FUNCTION_BLOCK "Stanowisko_KB2"	// FB 4
//wyglad lini
//
//
//||||   ||     ||||   ||||
//|Z||  |O||    |W |   |S |
//||||   ||     ||||   ||||
//      
//      ||||
//      |B||
//      ||||
//
//Gdzie:
//-W-Winda
//-S-Shuttle
//-Z-ZPA(Segbert)
//-O-Obrotnica
//-B-Banda Backup
//
//
//Wersja 1.1
//-Dodanie mo¿liwosci poboru palety z Bandy backup (pisanie w trakcie)
//
//
//
AUTHOR : Kng
NAME : KB2
VERSION : 0.1
VAR
  KB2_Wylot_2 : FB 33;
  KB2_Obrotnica : FB 35;
  KB2_Uzbrajanie : FB 10;
  KB2_Winda : FB 37;
END_VAR
BEGIN
NETWORK
TITLE =
//Ten Network celowo jest wolny
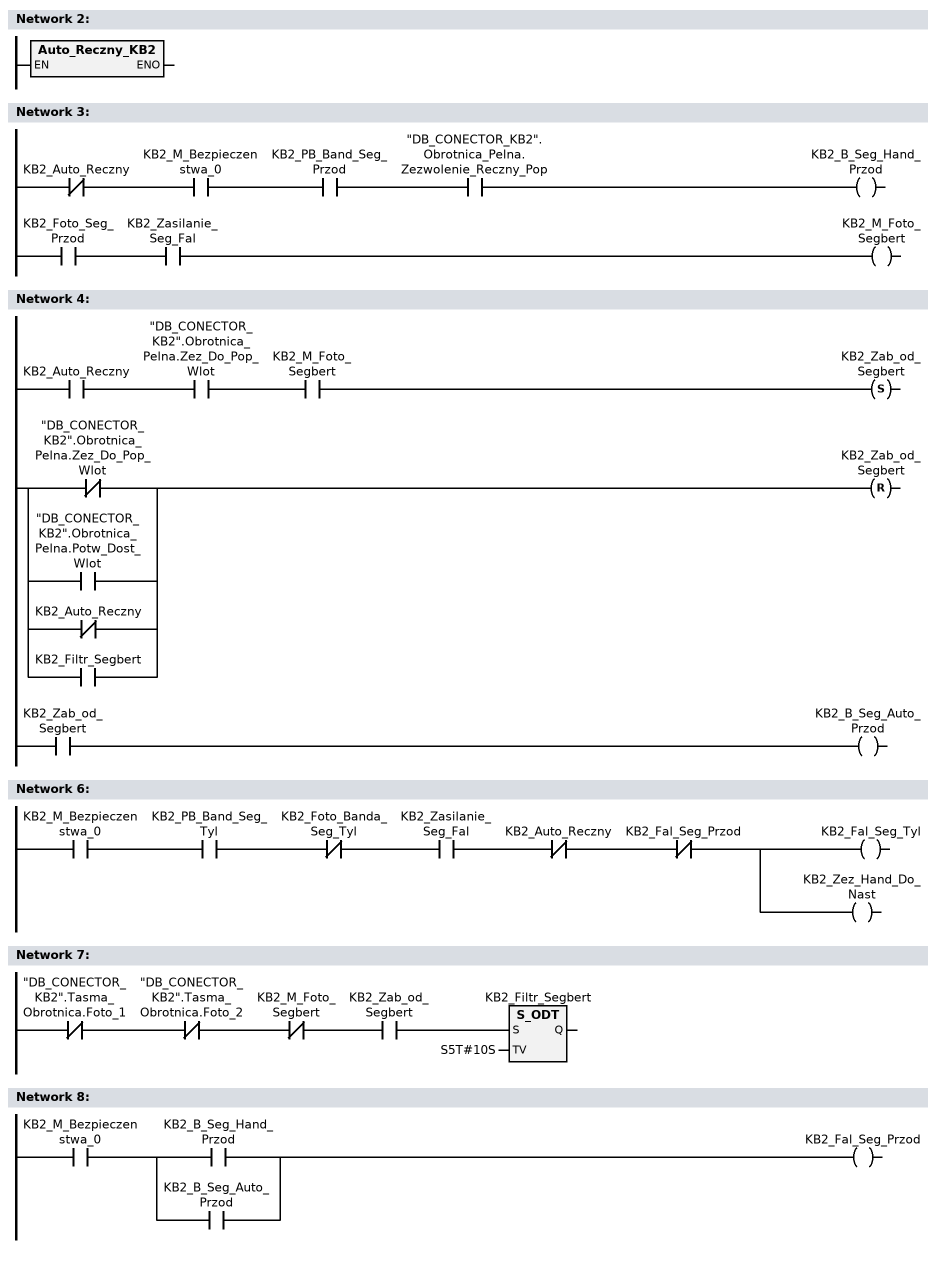
NETWORK
TITLE =
      CALL  "Auto_Reczny_KB2";
      NOP   0;
NETWORK
TITLE =
//Bity do Terminala
//
//Terminal_Palet                                   Szafa_Transport
//
//
//<-----------------------------------------------KB2_Fal_Seg_Przod (Q25.0)
//<-----------------------------------------------
//<-----------------------------------------------
//
//----------------------------------------------->KB2_Foto_Seg_Przod (I26.0)
//----------------------------------------------->
//----------------------------------------------->
//----------------------------------------------->
      AN    "KB2_Auto_Reczny";
      A     "KB2_M_Bezpieczenstwa_0";
      A     "KB2_PB_Band_Seg_Przod";
      A     "DB_CONECTOR_KB2".Obrotnica_Pelna.Zezwolenie_Reczny_Pop;
      =     "KB2_B_Seg_Hand_Przod";
//Wyjazd palety w automacie
      A     "KB2_Foto_Seg_Przod";
      A     "KB2_Zasilanie_Seg_Fal";
      =     "KB2_M_Foto_Segbert";
NETWORK
TITLE =
      A     "KB2_Auto_Reczny";
      A     "DB_CONECTOR_KB2".Obrotnica_Pelna.Zez_Do_Pop_Wlot;
      A     "KB2_M_Foto_Segbert";
      S     "KB2_Zab_od_Segbert";
      A(;
      ON    "DB_CONECTOR_KB2".Obrotnica_Pelna.Zez_Do_Pop_Wlot;
      O     "DB_CONECTOR_KB2".Obrotnica_Pelna.Potw_Dost_Wlot;
      ON    "KB2_Auto_Reczny";
      O     "KB2_Filtr_Segbert";
      );
      R     "KB2_Zab_od_Segbert";
      A     "KB2_Zab_od_Segbert";
      =     "KB2_B_Seg_Auto_Przod";
NETWORK
TITLE =
//Ten Network celowo jest wolny
NETWORK
TITLE =
//Segbert_Warunkowy tyl
      A     "KB2_M_Bezpieczenstwa_0";
      A     "KB2_PB_Band_Seg_Tyl";
      AN    "KB2_Foto_Banda_Seg_Tyl";
      A     "KB2_Zasilanie_Seg_Fal";
      AN    "KB2_Auto_Reczny";
      AN    "KB2_Fal_Seg_Przod";
      =     "KB2_Fal_Seg_Tyl";
      =     "KB2_Zez_Hand_Do_Nast";
NETWORK
TITLE =
      AN    "DB_CONECTOR_KB2".Tasma_Obrotnica.Foto_1;
      AN    "DB_CONECTOR_KB2".Tasma_Obrotnica.Foto_2;
      AN    "KB2_M_Foto_Segbert";
      A     "KB2_Zab_od_Segbert";
      L     S5T#10S;
      SD    "KB2_Filtr_Segbert";
      NOP   0;
      NOP   0;
      NOP   0;
      NOP   0;
NETWORK
TITLE =
//Jazda bandy Segbert do przodu
      A     "KB2_M_Bezpieczenstwa_0";
      A(;
      O     "KB2_B_Seg_Hand_Przod";
      O     "KB2_B_Seg_Auto_Przod";
      );
      =     "KB2_Fal_Seg_Przod";
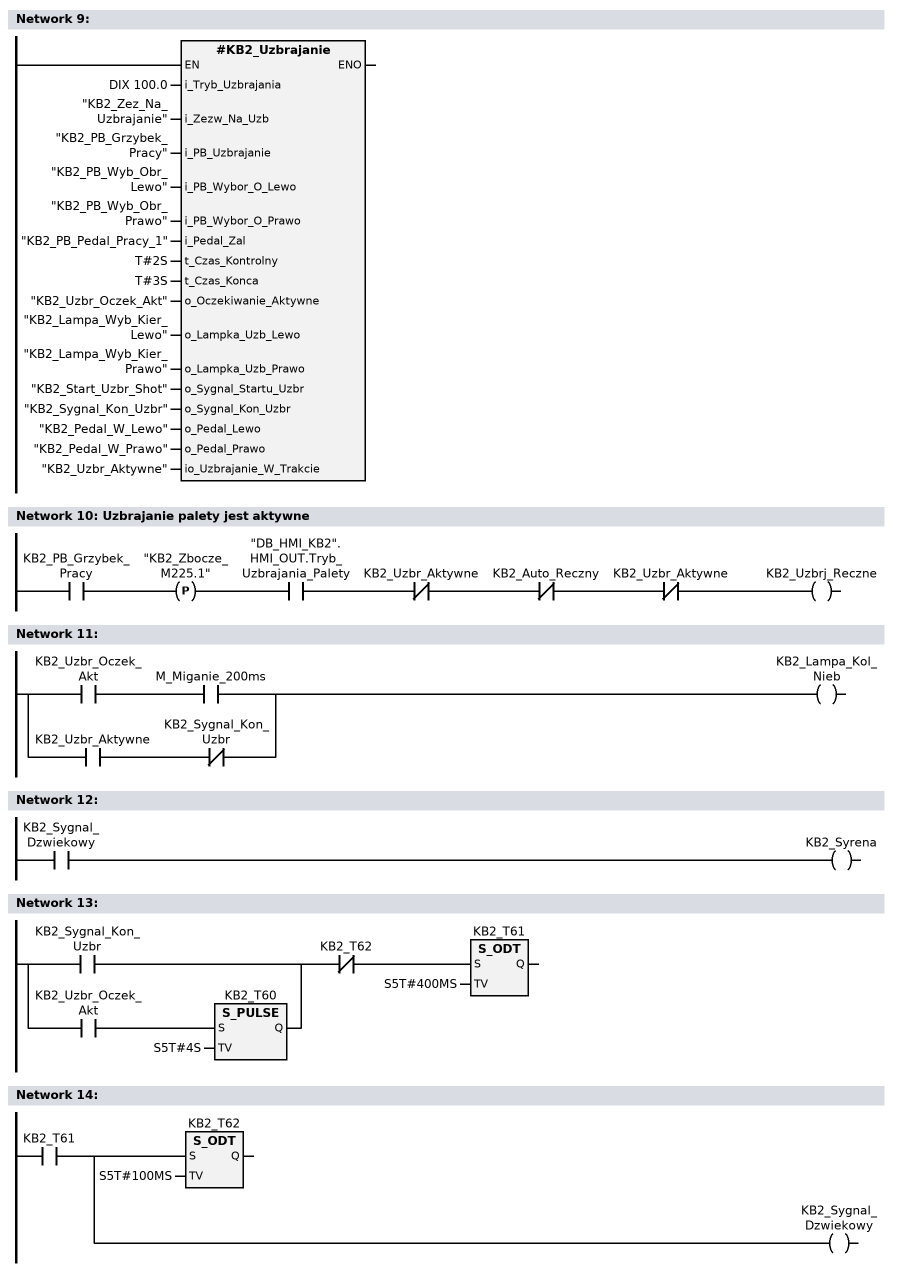
NETWORK
TITLE =
//Funkcja Uzbrajania
      CALL  #KB2_Uzbrajanie (
           i_Tryb_Uzbrajania        := DIX 100.0,
           i_Zezw_Na_Uzb            := "KB2_Zez_Na_Uzbrajanie",
           i_PB_Uzbrajanie          := "KB2_PB_Grzybek_Pracy",
           i_PB_Wybor_O_Lewo        := "KB2_PB_Wyb_Obr_Lewo",
           i_PB_Wybor_O_Prawo       := "KB2_PB_Wyb_Obr_Prawo",
           i_Pedal_Zal              := "KB2_PB_Pedal_Pracy_1",
           t_Czas_Kontrolny         := T#2S,
           t_Czas_Konca             := T#3S,
           o_Oczekiwanie_Aktywne    := "KB2_Uzbr_Oczek_Akt",
           o_Lampka_Uzb_Lewo        := "KB2_Lampa_Wyb_Kier_Lewo",
           o_Lampka_Uzb_Prawo       := "KB2_Lampa_Wyb_Kier_Prawo",
           o_Sygnal_Startu_Uzbr     := "KB2_Start_Uzbr_Shot",
           o_Sygnal_Kon_Uzbr        := "KB2_Sygnal_Kon_Uzbr",
           o_Pedal_Lewo             := "KB2_Pedal_W_Lewo",
           o_Pedal_Prawo            := "KB2_Pedal_W_Prawo",
           io_Uzbrajanie_W_Trakcie  := "KB2_Uzbr_Aktywne");
NETWORK
TITLE = Uzbrajanie palety jest aktywne
//Uzbrajanie reczne 
      A     "KB2_PB_Grzybek_Pracy";
      FP    "KB2_Zbocze_M225.1";
      A     "DB_HMI_KB2".HMI_OUT.Tryb_Uzbrajania_Palety;
      AN    "KB2_Uzbr_Aktywne";
      AN    "KB2_Auto_Reczny";
      AN    "KB2_Uzbr_Aktywne";
      =     "KB2_Uzbrj_Reczne";
NETWORK
TITLE =
//Lampka uzbrajania
//
      A     "KB2_Uzbr_Oczek_Akt";
      A     "M_Miganie_200ms";
      O;
      A     "KB2_Uzbr_Aktywne";
      AN    "KB2_Sygnal_Kon_Uzbr";
      =     "KB2_Lampa_Kol_Nieb";
NETWORK
TITLE =
//Sygnal dzwiekowy uzbrajania
//
      A     "KB2_Sygnal_Dzwiekowy";
      =     "KB2_Syrena";
NETWORK
TITLE =
//Tworzenie dzwieku
      A(;
      O     "KB2_Sygnal_Kon_Uzbr";
      O(;
      A     "KB2_Uzbr_Oczek_Akt";
      L     S5T#4S;
      SP    "KB2_T60";
      NOP   0;
      NOP   0;
      NOP   0;
      A     "KB2_T60";
      );
      );
      AN    "KB2_T62";
      L     S5T#400MS;
      SD    "KB2_T61";
      NOP   0;
      NOP   0;
      NOP   0;
      NOP   0;
NETWORK
TITLE =
      A     "KB2_T61";
      =     L 0.0;
      A     L 0.0;
      L     S5T#100MS;
      SD    "KB2_T62";
      NOP   0;
      NOP   0;
      NOP   0;
      NOP   0;
      A     L 0.0;
      BLD   102;
      =     "KB2_Sygnal_Dzwiekowy";
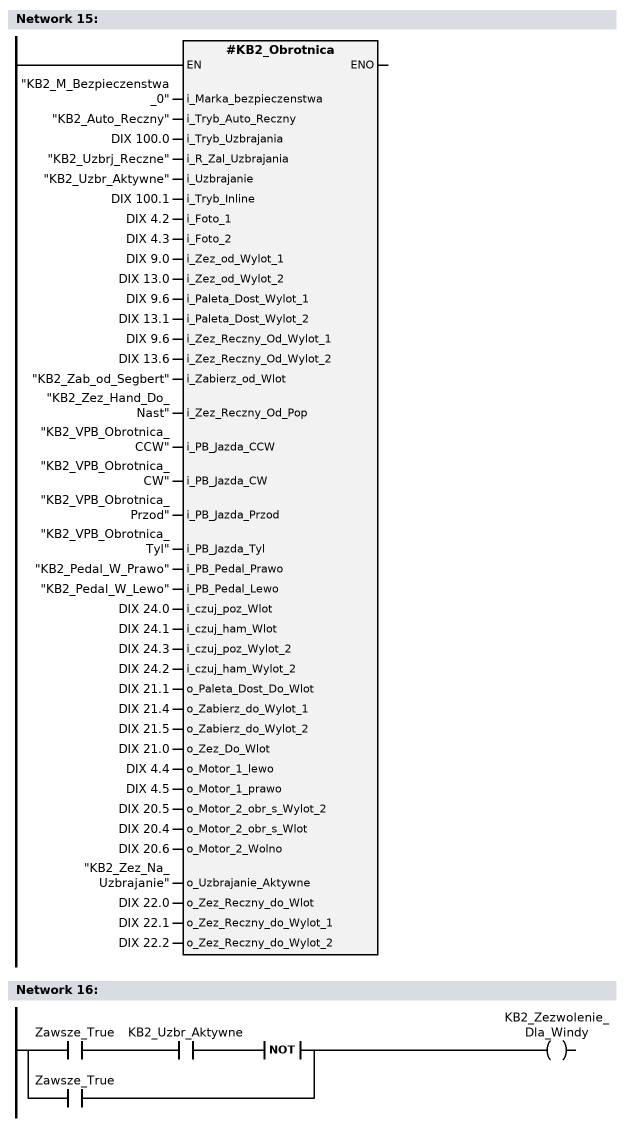
NETWORK
TITLE =
//Obrotnica z funkcja uzbrajania
      CALL  #KB2_Obrotnica (
           i_Marka_bezpieczenstwa   := "KB2_M_Bezpieczenstwa_0",
           i_Tryb_Auto_Reczny       := "KB2_Auto_Reczny",
           i_Tryb_Uzbrajania        := DIX 100.0,
           i_R_Zal_Uzbrajania       := "KB2_Uzbrj_Reczne",
           i_Uzbrajanie             := "KB2_Uzbr_Aktywne",
           i_Tryb_Inline            := DIX 100.1,
           i_Foto_1                 := DIX 4.2,
           i_Foto_2                 := DIX 4.3,
           i_Zez_od_Wylot_1         := DIX 9.0,
           i_Zez_od_Wylot_2         := DIX 13.0,
           i_Paleta_Dost_Wylot_1    := DIX 9.6,
           i_Paleta_Dost_Wylot_2    := DIX 13.1,
           i_Zez_Reczny_Od_Wylot_1  := DIX 9.6,
           i_Zez_Reczny_Od_Wylot_2  := DIX 13.6,
           i_Zabierz_od_Wlot        := "KB2_Zab_od_Segbert",
           i_Zez_Reczny_Od_Pop      := "KB2_Zez_Hand_Do_Nast",
           i_PB_Jazda_CCW           := "KB2_VPB_Obrotnica_CCW",
           i_PB_Jazda_CW            := "KB2_VPB_Obrotnica_CW",
           i_PB_Jazda_Przod         := "KB2_VPB_Obrotnica_Przod",
           i_PB_Jazda_Tyl           := "KB2_VPB_Obrotnica_Tyl",
           i_PB_Pedal_Prawo         := "KB2_Pedal_W_Prawo",
           i_PB_Pedal_Lewo          := "KB2_Pedal_W_Lewo",
           i_czuj_poz_Wlot          := DIX 24.0,
           i_czuj_ham_Wlot          := DIX 24.1,
           i_czuj_poz_Wylot_2       := DIX 24.3,
           i_czuj_ham_Wylot_2       := DIX 24.2,
           o_Paleta_Dost_Do_Wlot    := DIX 21.1,
           o_Zabierz_do_Wylot_1     := DIX 21.4,
           o_Zabierz_do_Wylot_2     := DIX 21.5,
           o_Zez_Do_Wlot            := DIX 21.0,
           o_Motor_1_lewo           := DIX 4.4,
           o_Motor_1_prawo          := DIX 4.5,
           o_Motor_2_obr_s_Wylot_2  := DIX 20.5,
           o_Motor_2_obr_s_Wlot     := DIX 20.4,
           o_Motor_2_Wolno          := DIX 20.6,
           o_Uzbrajanie_Aktywne     := "KB2_Zez_Na_Uzbrajanie",
           o_Zez_Reczny_do_Wlot     := DIX 22.0,
           o_Zez_Reczny_do_Wylot_1  := DIX 22.1,
           o_Zez_Reczny_do_Wylot_2  := DIX 22.2);
NETWORK
TITLE =
      A     "Zawsze_True";
      A     "KB2_Uzbr_Aktywne";
      NOT;
      O     "Zawsze_True";
      =     "KB2_Zezwolenie_Dla_Windy";
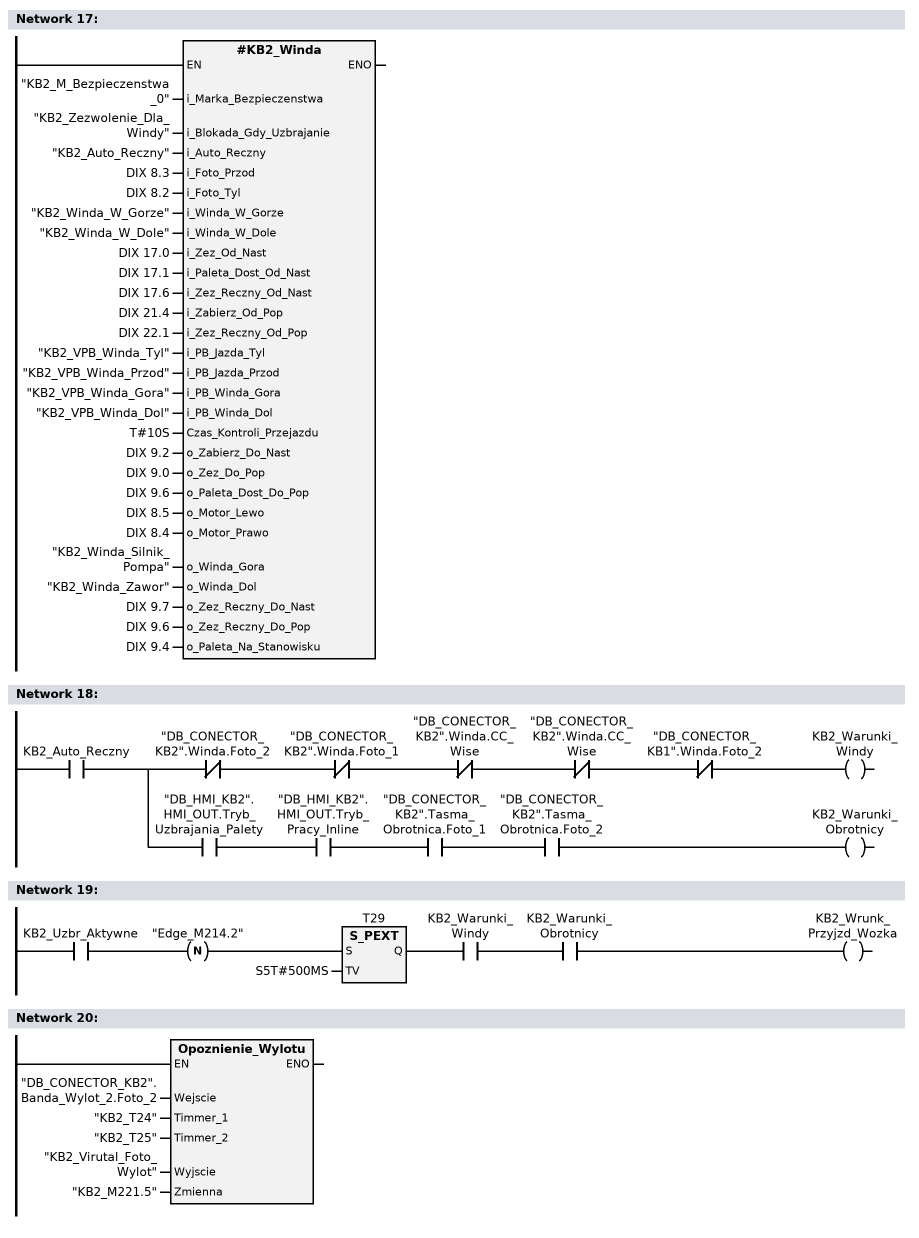
NETWORK
TITLE =
//Winda
      CALL  #KB2_Winda (
           i_Marka_Bezpieczenstwa   := "KB2_M_Bezpieczenstwa_0",
           i_Blokada_Gdy_Uzbrajanie := "KB2_Zezwolenie_Dla_Windy",
           i_Auto_Reczny            := "KB2_Auto_Reczny",
           i_Foto_Przod             := DIX 8.3,
           i_Foto_Tyl               := DIX 8.2,
           i_Winda_W_Gorze          := "KB2_Winda_W_Gorze",
           i_Winda_W_Dole           := "KB2_Winda_W_Dole",
           i_Zez_Od_Nast            := DIX 17.0,
           i_Paleta_Dost_Od_Nast    := DIX 17.1,
           i_Zez_Reczny_Od_Nast     := DIX 17.6,
           i_Zabierz_Od_Pop         := DIX 21.4,
           i_Zez_Reczny_Od_Pop      := DIX 22.1,
           i_PB_Jazda_Tyl           := "KB2_VPB_Winda_Tyl",
           i_PB_Jazda_Przod         := "KB2_VPB_Winda_Przod",
           i_PB_Winda_Gora          := "KB2_VPB_Winda_Gora",
           i_PB_Winda_Dol           := "KB2_VPB_Winda_Dol",
           Czas_Kontroli_Przejazdu  := T#10S,
           o_Zabierz_Do_Nast        := DIX 9.2,
           o_Zez_Do_Pop             := DIX 9.0,
           o_Paleta_Dost_Do_Pop     := DIX 9.6,
           o_Motor_Lewo             := DIX 8.5,
           o_Motor_Prawo            := DIX 8.4,
           o_Winda_Gora             := "KB2_Winda_Silnik_Pompa",
           o_Winda_Dol              := "KB2_Winda_Zawor",
           o_Zez_Reczny_Do_Nast     := DIX 9.7,
           o_Zez_Reczny_Do_Pop      := DIX 9.6,
           o_Paleta_Na_Stanowisku   := DIX 9.4);
NETWORK
TITLE =
//Warunkowa jazda wozka gdy konczone jest owijanie
//Warunki windy.
      A     "KB2_Auto_Reczny";
      =     L 0.0;
      A     L 0.0;
      AN    "DB_CONECTOR_KB2".Winda.Foto_2;
      AN    "DB_CONECTOR_KB2".Winda.Foto_1;
      AN    "DB_CONECTOR_KB2".Winda.CC_Wise;
      AN    "DB_CONECTOR_KB2".Winda.CC_Wise;
      AN    "DB_CONECTOR_KB1".Winda.Foto_2;
      =     "KB2_Warunki_Windy";
      A     L 0.0;
      A     "DB_HMI_KB2".HMI_OUT.Tryb_Uzbrajania_Palety;
      A     "DB_HMI_KB2".HMI_OUT.Tryb_Pracy_Inline;
      A     "DB_CONECTOR_KB2".Tasma_Obrotnica.Foto_1;
      A     "DB_CONECTOR_KB2".Tasma_Obrotnica.Foto_2;
      =     "KB2_Warunki_Obrotnicy";
NETWORK
TITLE =
//Warunki obrotnicy
      A(;
      A     "KB2_Uzbr_Aktywne";
      FN    "Edge_M214.2";
      L     S5T#500MS;
      SE    "T29";
      NOP   0;
      NOP   0;
      NOP   0;
      A     "T29";
      );
      A     "KB2_Warunki_Windy";
      A     "KB2_Warunki_Obrotnicy";
      =     "KB2_Wrunk_Przyjzd_Wozka";
NETWORK
TITLE =
//Opoznienie wylotu
      CALL  "Opoznienie_Wylotu" (
           Wejscie                  := "DB_CONECTOR_KB2".Banda_Wylot_2.Foto_2,
           Timmer_1                 := "KB2_T24",
           Timmer_2                 := "KB2_T25",
           Wyjscie                  := "KB2_Virutal_Foto_Wylot",
           Zmienna                  := "KB2_M221.5");
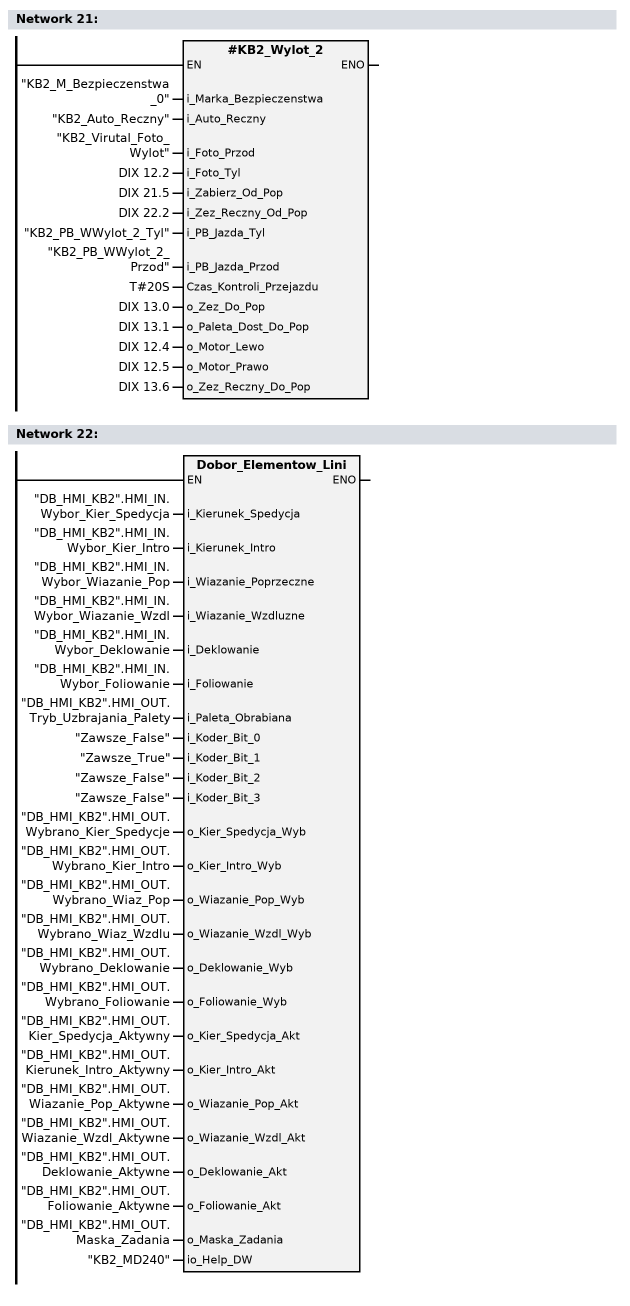
NETWORK
TITLE =
//Banda Wylot 2
      CALL  #KB2_Wylot_2 (
           i_Marka_Bezpieczenstwa   := "KB2_M_Bezpieczenstwa_0",
           i_Auto_Reczny            := "KB2_Auto_Reczny",
           i_Foto_Przod             := "KB2_Virutal_Foto_Wylot",
           i_Foto_Tyl               := DIX 12.2,
           i_Zabierz_Od_Pop         := DIX 21.5,
           i_Zez_Reczny_Od_Pop      := DIX 22.2,
           i_PB_Jazda_Tyl           := "KB2_PB_WWylot_2_Tyl",
           i_PB_Jazda_Przod         := "KB2_PB_WWylot_2_Przod",
           Czas_Kontroli_Przejazdu  := T#20S,
           o_Zez_Do_Pop             := DIX 13.0,
           o_Paleta_Dost_Do_Pop     := DIX 13.1,
           o_Motor_Lewo             := DIX 12.4,
           o_Motor_Prawo            := DIX 12.5,
           o_Zez_Reczny_Do_Pop      := DIX 13.6);
NETWORK
TITLE =
//fc400. Kod kolbus 2 to 2 .
      CALL  "Dobor_Elementow_Lini" (
           i_Kierunek_Spedycja      := "DB_HMI_KB2".HMI_IN.Wybor_Kier_Spedycja,
           i_Kierunek_Intro         := "DB_HMI_KB2".HMI_IN.Wybor_Kier_Intro,
           i_Wiazanie_Poprzeczne    := "DB_HMI_KB2".HMI_IN.Wybor_Wiazanie_Pop,
           i_Wiazanie_Wzdluzne      := "DB_HMI_KB2".HMI_IN.Wybor_Wiazanie_Wzdl,
           i_Deklowanie             := "DB_HMI_KB2".HMI_IN.Wybor_Deklowanie,
           i_Foliowanie             := "DB_HMI_KB2".HMI_IN.Wybor_Foliowanie,
           i_Paleta_Obrabiana       := "DB_HMI_KB2".HMI_OUT.Tryb_Uzbrajania_Palety,
           i_Koder_Bit_0            := "Zawsze_False",
           i_Koder_Bit_1            := "Zawsze_True",
           i_Koder_Bit_2            := "Zawsze_False",
           i_Koder_Bit_3            := "Zawsze_False",
           o_Kier_Spedycja_Wyb      := "DB_HMI_KB2".HMI_OUT.Wybrano_Kier_Spedycje,
           o_Kier_Intro_Wyb         := "DB_HMI_KB2".HMI_OUT.Wybrano_Kier_Intro,
           o_Wiazanie_Pop_Wyb       := "DB_HMI_KB2".HMI_OUT.Wybrano_Wiaz_Pop,
           o_Wiazanie_Wzdl_Wyb      := "DB_HMI_KB2".HMI_OUT.Wybrano_Wiaz_Wzdlu,
           o_Deklowanie_Wyb         := "DB_HMI_KB2".HMI_OUT.Wybrano_Deklowanie,
           o_Foliowanie_Wyb         := "DB_HMI_KB2".HMI_OUT.Wybrano_Foliowanie,
           o_Kier_Spedycja_Akt      := "DB_HMI_KB2".HMI_OUT.Kier_Spedycja_Aktywny,
           o_Kier_Intro_Akt         := "DB_HMI_KB2".HMI_OUT.Kierunek_Intro_Aktywny,
           o_Wiazanie_Pop_Akt       := "DB_HMI_KB2".HMI_OUT.Wiazanie_Pop_Aktywne,
           o_Wiazanie_Wzdl_Akt      := "DB_HMI_KB2".HMI_OUT.Wiazanie_Wzdl_Aktywne,
           o_Deklowanie_Akt         := "DB_HMI_KB2".HMI_OUT.Deklowanie_Aktywne,
           o_Foliowanie_Akt         := "DB_HMI_KB2".HMI_OUT.Foliowanie_Aktywne,
           o_Maska_Zadania          := "DB_HMI_KB2".HMI_OUT.Maska_Zadania,
           io_Help_DW               := "KB2_MD240");
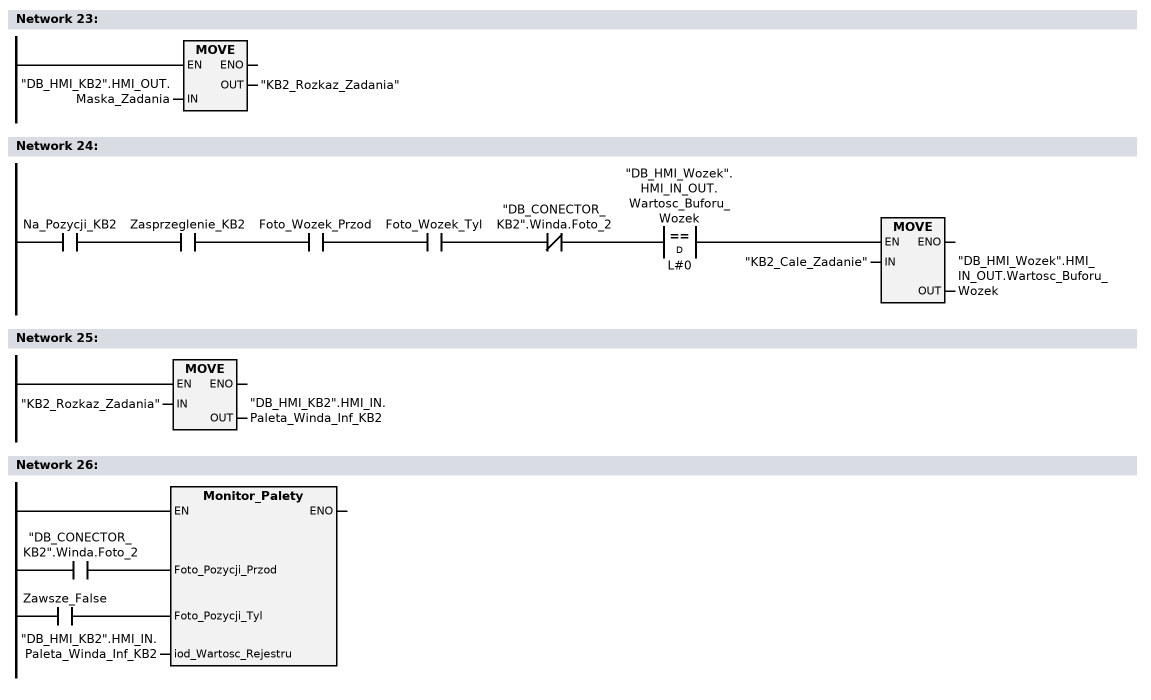
NETWORK
TITLE =
//Przeslanie maski do starszego slowa
      L     "DB_HMI_KB2".HMI_OUT.Maska_Zadania;
      T     "KB2_Rozkaz_Zadania";
      NOP   0;
NETWORK
TITLE =
//To jest wozek
//
      A     "Na_Pozycji_KB2";
      A     "Zasprzeglenie_KB2";
      A     "Foto_Wozek_Przod";
      A     "Foto_Wozek_Tyl";
      AN    "DB_CONECTOR_KB2".Winda.Foto_2;
      A(;
      L     "DB_HMI_Wozek".HMI_IN_OUT.Wartosc_Buforu_Wozek;
      L     L#0;
      ==D;
      );
      JNB   _001;
      L     "KB2_Cale_Zadanie";
      T     "DB_HMI_Wozek".HMI_IN_OUT.Wartosc_Buforu_Wozek;
_001: NOP   0;
NETWORK
TITLE =
      L     "KB2_Rozkaz_Zadania";
      T     "DB_HMI_KB2".HMI_IN.Paleta_Winda_Inf_KB2;
      NOP   0;
NETWORK
TITLE =
      A     "DB_CONECTOR_KB2".Winda.Foto_2;
      =     L 0.0;
      BLD   103;
      A     "Zawsze_False";
      =     L 0.1;
      BLD   103;
      CALL  "Monitor_Palety" (
           Foto_Pozycji_Przod       := L 0.0,
           Foto_Pozycji_Tyl         := L 0.1,
           iod_Wartosc_Rejestru     := "DB_HMI_KB2".HMI_IN.Paleta_Winda_Inf_KB2);
      NOP   0;
END_FUNCTION_BLOCK

FUNCTION_BLOCK "Stan_Intro_Odbieranie"	// FB 6
//Stanowisko intro Odbieranie
//Linia zlozona z 5 band odbierajacych
//
//
//BW B2 B3 B4 B4 B6
//===>
//
//5 band kierunek zwyczajny
VERSION : 0.1
VAR
  Banda_2 : FB 33;
  Banda_3 : FB 33;
  Banda_4 : FB 33;
  Banda_5 : FB 33;
  Banda_6 : FB 33;
END_VAR
VAR_TEMP
  help_bit_1 : BOOL ;
  Help_Reczny_Przod : BOOL ;
  Help_Reczny_Tyl : BOOL ;
END_VAR
BEGIN
NETWORK
TITLE =
//Ten Network celowo jest wolny
NETWORK
TITLE =
//Banda poprzednia jest wozek jezdny
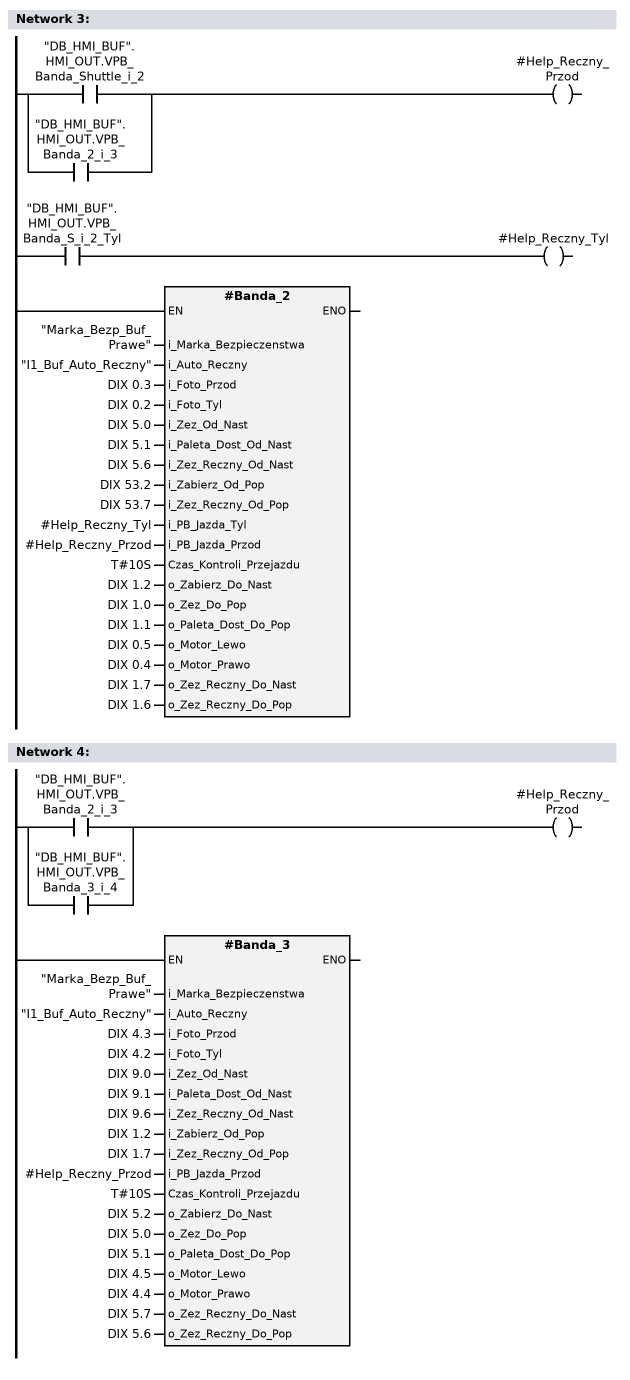
NETWORK
TITLE =
//Banda 2
      O     "DB_HMI_BUF".HMI_OUT.VPB_Banda_Shuttle_i_2;
      O     "DB_HMI_BUF".HMI_OUT.VPB_Banda_2_i_3;
      =     #Help_Reczny_Przod;
      O     "DB_HMI_BUF".HMI_OUT.VPB_Banda_S_i_2_Tyl;
      =     #Help_Reczny_Tyl;
      CALL  #Banda_2 (
           i_Marka_Bezpieczenstwa   := "Marka_Bezp_Buf_Prawe",
           i_Auto_Reczny            := "I1_Buf_Auto_Reczny",
           i_Foto_Przod             := DIX 0.3,
           i_Foto_Tyl               := DIX 0.2,
           i_Zez_Od_Nast            := DIX 5.0,
           i_Paleta_Dost_Od_Nast    := DIX 5.1,
           i_Zez_Reczny_Od_Nast     := DIX 5.6,
           i_Zabierz_Od_Pop         := DIX 53.2,
           i_Zez_Reczny_Od_Pop      := DIX 53.7,
           i_PB_Jazda_Tyl           := #Help_Reczny_Tyl,
           i_PB_Jazda_Przod         := #Help_Reczny_Przod,
           Czas_Kontroli_Przejazdu  := T#10S,
           o_Zabierz_Do_Nast        := DIX 1.2,
           o_Zez_Do_Pop             := DIX 1.0,
           o_Paleta_Dost_Do_Pop     := DIX 1.1,
           o_Motor_Lewo             := DIX 0.5,
           o_Motor_Prawo            := DIX 0.4,
           o_Zez_Reczny_Do_Nast     := DIX 1.7,
           o_Zez_Reczny_Do_Pop      := DIX 1.6);
NETWORK
TITLE =
//Banda 3
      O     "DB_HMI_BUF".HMI_OUT.VPB_Banda_2_i_3;
      O     "DB_HMI_BUF".HMI_OUT.VPB_Banda_3_i_4;
      =     #Help_Reczny_Przod;
      CALL  #Banda_3 (
           i_Marka_Bezpieczenstwa   := "Marka_Bezp_Buf_Prawe",
           i_Auto_Reczny            := "I1_Buf_Auto_Reczny",
           i_Foto_Przod             := DIX 4.3,
           i_Foto_Tyl               := DIX 4.2,
           i_Zez_Od_Nast            := DIX 9.0,
           i_Paleta_Dost_Od_Nast    := DIX 9.1,
           i_Zez_Reczny_Od_Nast     := DIX 9.6,
           i_Zabierz_Od_Pop         := DIX 1.2,
           i_Zez_Reczny_Od_Pop      := DIX 1.7,
           i_PB_Jazda_Przod         := #Help_Reczny_Przod,
           Czas_Kontroli_Przejazdu  := T#10S,
           o_Zabierz_Do_Nast        := DIX 5.2,
           o_Zez_Do_Pop             := DIX 5.0,
           o_Paleta_Dost_Do_Pop     := DIX 5.1,
           o_Motor_Lewo             := DIX 4.5,
           o_Motor_Prawo            := DIX 4.4,
           o_Zez_Reczny_Do_Nast     := DIX 5.7,
           o_Zez_Reczny_Do_Pop      := DIX 5.6);
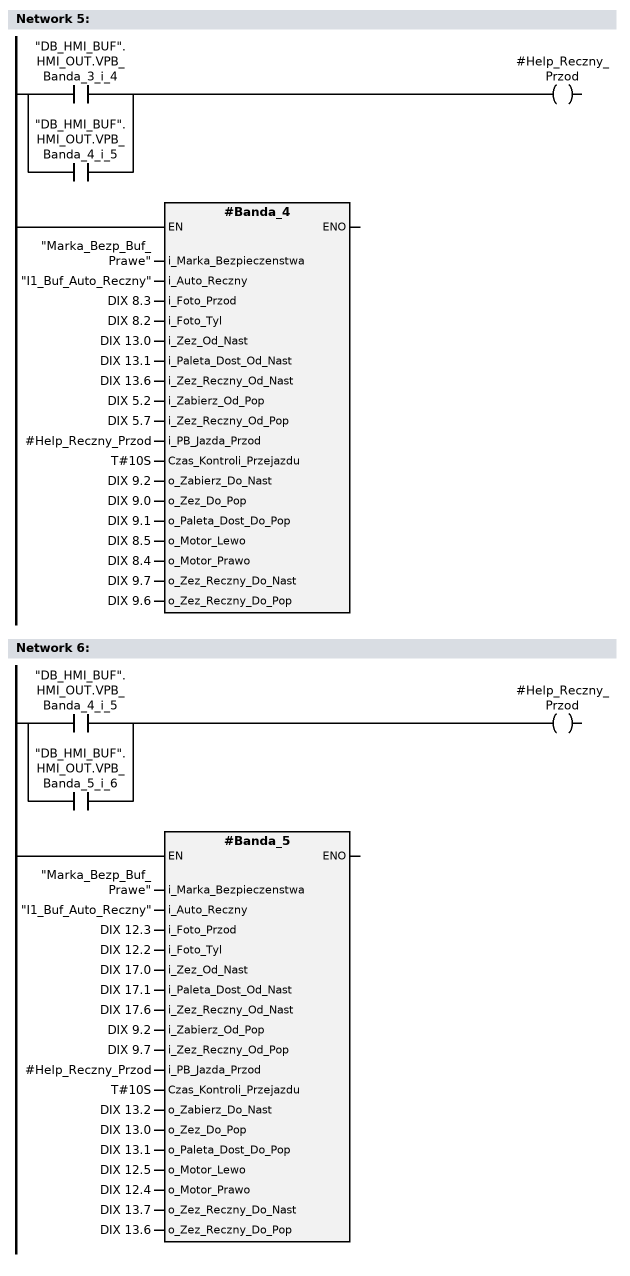
NETWORK
TITLE =
//Banda 4
      O     "DB_HMI_BUF".HMI_OUT.VPB_Banda_3_i_4;
      O     "DB_HMI_BUF".HMI_OUT.VPB_Banda_4_i_5;
      =     #Help_Reczny_Przod;
      CALL  #Banda_4 (
           i_Marka_Bezpieczenstwa   := "Marka_Bezp_Buf_Prawe",
           i_Auto_Reczny            := "I1_Buf_Auto_Reczny",
           i_Foto_Przod             := DIX 8.3,
           i_Foto_Tyl               := DIX 8.2,
           i_Zez_Od_Nast            := DIX 13.0,
           i_Paleta_Dost_Od_Nast    := DIX 13.1,
           i_Zez_Reczny_Od_Nast     := DIX 13.6,
           i_Zabierz_Od_Pop         := DIX 5.2,
           i_Zez_Reczny_Od_Pop      := DIX 5.7,
           i_PB_Jazda_Przod         := #Help_Reczny_Przod,
           Czas_Kontroli_Przejazdu  := T#10S,
           o_Zabierz_Do_Nast        := DIX 9.2,
           o_Zez_Do_Pop             := DIX 9.0,
           o_Paleta_Dost_Do_Pop     := DIX 9.1,
           o_Motor_Lewo             := DIX 8.5,
           o_Motor_Prawo            := DIX 8.4,
           o_Zez_Reczny_Do_Nast     := DIX 9.7,
           o_Zez_Reczny_Do_Pop      := DIX 9.6);
NETWORK
TITLE =
//Banda 5
      O     "DB_HMI_BUF".HMI_OUT.VPB_Banda_4_i_5;
      O     "DB_HMI_BUF".HMI_OUT.VPB_Banda_5_i_6;
      =     #Help_Reczny_Przod;
      CALL  #Banda_5 (
           i_Marka_Bezpieczenstwa   := "Marka_Bezp_Buf_Prawe",
           i_Auto_Reczny            := "I1_Buf_Auto_Reczny",
           i_Foto_Przod             := DIX 12.3,
           i_Foto_Tyl               := DIX 12.2,
           i_Zez_Od_Nast            := DIX 17.0,
           i_Paleta_Dost_Od_Nast    := DIX 17.1,
           i_Zez_Reczny_Od_Nast     := DIX 17.6,
           i_Zabierz_Od_Pop         := DIX 9.2,
           i_Zez_Reczny_Od_Pop      := DIX 9.7,
           i_PB_Jazda_Przod         := #Help_Reczny_Przod,
           Czas_Kontroli_Przejazdu  := T#10S,
           o_Zabierz_Do_Nast        := DIX 13.2,
           o_Zez_Do_Pop             := DIX 13.0,
           o_Paleta_Dost_Do_Pop     := DIX 13.1,
           o_Motor_Lewo             := DIX 12.5,
           o_Motor_Prawo            := DIX 12.4,
           o_Zez_Reczny_Do_Nast     := DIX 13.7,
           o_Zez_Reczny_Do_Pop      := DIX 13.6);
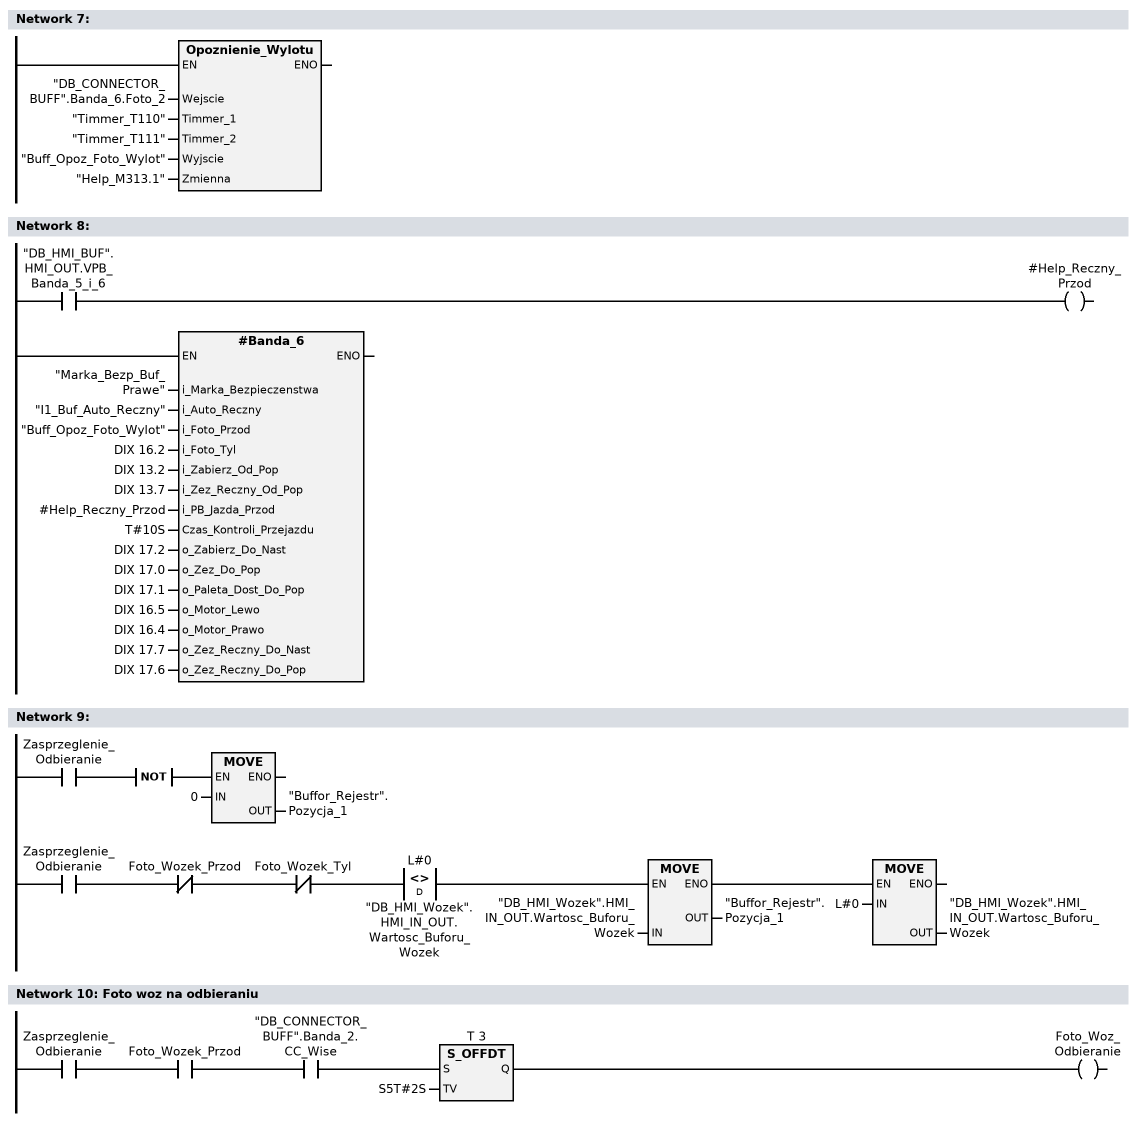
NETWORK
TITLE =
      CALL  "Opoznienie_Wylotu" (
           Wejscie                  := "DB_CONNECTOR_BUFF".Banda_6.Foto_2,
           Timmer_1                 := "Timmer_T110",
           Timmer_2                 := "Timmer_T111",
           Wyjscie                  := "Buff_Opoz_Foto_Wylot",
           Zmienna                  := "Help_M313.1");
NETWORK
TITLE =
//Banda 6
      O     "DB_HMI_BUF".HMI_OUT.VPB_Banda_5_i_6;
      =     #Help_Reczny_Przod;
      CALL  #Banda_6 (
           i_Marka_Bezpieczenstwa   := "Marka_Bezp_Buf_Prawe",
           i_Auto_Reczny            := "I1_Buf_Auto_Reczny",
           i_Foto_Przod             := "Buff_Opoz_Foto_Wylot",
           i_Foto_Tyl               := DIX 16.2,
           i_Zabierz_Od_Pop         := DIX 13.2,
           i_Zez_Reczny_Od_Pop      := DIX 13.7,
           i_PB_Jazda_Przod         := #Help_Reczny_Przod,
           Czas_Kontroli_Przejazdu  := T#10S,
           o_Zabierz_Do_Nast        := DIX 17.2,
           o_Zez_Do_Pop             := DIX 17.0,
           o_Paleta_Dost_Do_Pop     := DIX 17.1,
           o_Motor_Lewo             := DIX 16.5,
           o_Motor_Prawo            := DIX 16.4,
           o_Zez_Reczny_Do_Nast     := DIX 17.7,
           o_Zez_Reczny_Do_Pop      := DIX 17.6);
NETWORK
TITLE =
      A     "Zasprzeglenie_Odbieranie";
      =     L 1.0;
      A(;
      A     L 1.0;
      AN    "Foto_Wozek_Przod";
      AN    "Foto_Wozek_Tyl";
      A(;
      L     L#0;
      L     "DB_HMI_Wozek".HMI_IN_OUT.Wartosc_Buforu_Wozek;
      <>D;
      );
      JNB   _001;
      L     "DB_HMI_Wozek".HMI_IN_OUT.Wartosc_Buforu_Wozek;
      T     "Buffor_Rejestr".Pozycja_1;
      SET;
      SAVE;
      CLR;
_001: A     BR;
      );
      JNB   _002;
      L     L#0;
      T     "DB_HMI_Wozek".HMI_IN_OUT.Wartosc_Buforu_Wozek;
_002: NOP   0;
      A     L 1.0;
      NOT;
      JNB   _003;
      L     0;
      T     "Buffor_Rejestr".Pozycja_1;
_003: NOP   0;
NETWORK
TITLE = Foto woz na odbieraniu
      A     "Zasprzeglenie_Odbieranie";
      A     "Foto_Wozek_Przod";
      A     "DB_CONNECTOR_BUFF".Banda_2.CC_Wise;
      L     S5T#2S;
      SF    T 3;
      NOP   0;
      NOP   0;
      NOP   0;
      A     T 3;
      =     "Foto_Woz_Odbieranie";
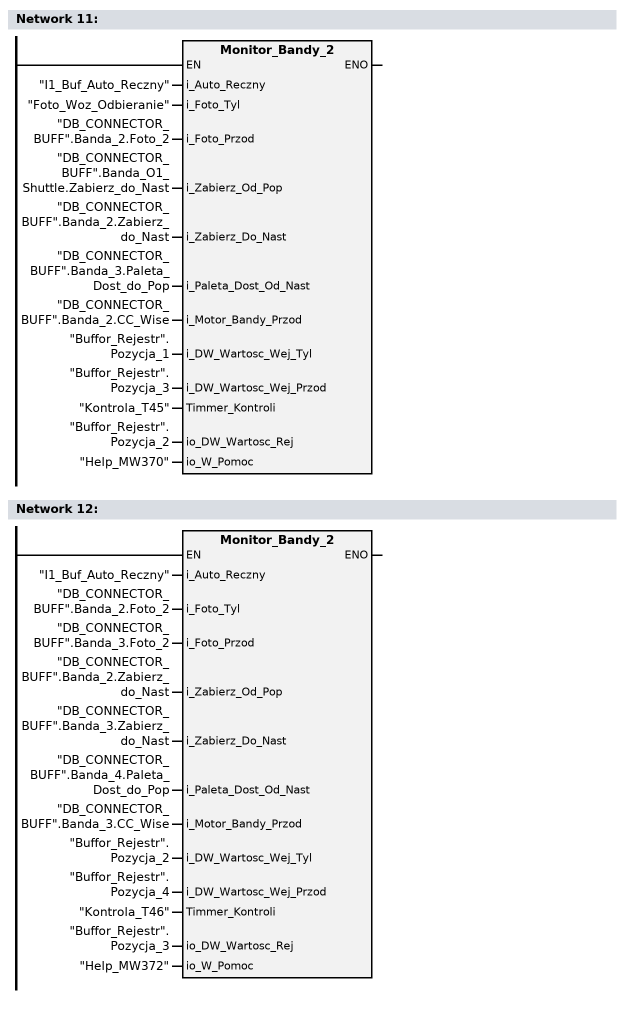
NETWORK
TITLE =
//Monitoring band 2
      CALL  "Monitor_Bandy_2" (
           i_Auto_Reczny            := "I1_Buf_Auto_Reczny",
           i_Foto_Tyl               := "Foto_Woz_Odbieranie",
           i_Foto_Przod             := "DB_CONNECTOR_BUFF".Banda_2.Foto_2,
           i_Zabierz_Od_Pop         := "DB_CONNECTOR_BUFF".Banda_O1_Shuttle.Zabierz_do_Nast,
           i_Zabierz_Do_Nast        := "DB_CONNECTOR_BUFF".Banda_2.Zabierz_do_Nast,
           i_Paleta_Dost_Od_Nast    := "DB_CONNECTOR_BUFF".Banda_3.Paleta_Dost_do_Pop,
           i_Motor_Bandy_Przod      := "DB_CONNECTOR_BUFF".Banda_2.CC_Wise,
           i_DW_Wartosc_Wej_Tyl     := "Buffor_Rejestr".Pozycja_1,
           i_DW_Wartosc_Wej_Przod   := "Buffor_Rejestr".Pozycja_3,
           Timmer_Kontroli          := "Kontrola_T45",
           io_DW_Wartosc_Rej        := "Buffor_Rejestr".Pozycja_2,
           io_W_Pomoc               := "Help_MW370");
NETWORK
TITLE =
//Monitoring band 3
      CALL  "Monitor_Bandy_2" (
           i_Auto_Reczny            := "I1_Buf_Auto_Reczny",
           i_Foto_Tyl               := "DB_CONNECTOR_BUFF".Banda_2.Foto_2,
           i_Foto_Przod             := "DB_CONNECTOR_BUFF".Banda_3.Foto_2,
           i_Zabierz_Od_Pop         := "DB_CONNECTOR_BUFF".Banda_2.Zabierz_do_Nast,
           i_Zabierz_Do_Nast        := "DB_CONNECTOR_BUFF".Banda_3.Zabierz_do_Nast,
           i_Paleta_Dost_Od_Nast    := "DB_CONNECTOR_BUFF".Banda_4.Paleta_Dost_do_Pop,
           i_Motor_Bandy_Przod      := "DB_CONNECTOR_BUFF".Banda_3.CC_Wise,
           i_DW_Wartosc_Wej_Tyl     := "Buffor_Rejestr".Pozycja_2,
           i_DW_Wartosc_Wej_Przod   := "Buffor_Rejestr".Pozycja_4,
           Timmer_Kontroli          := "Kontrola_T46",
           io_DW_Wartosc_Rej        := "Buffor_Rejestr".Pozycja_3,
           io_W_Pomoc               := "Help_MW372");
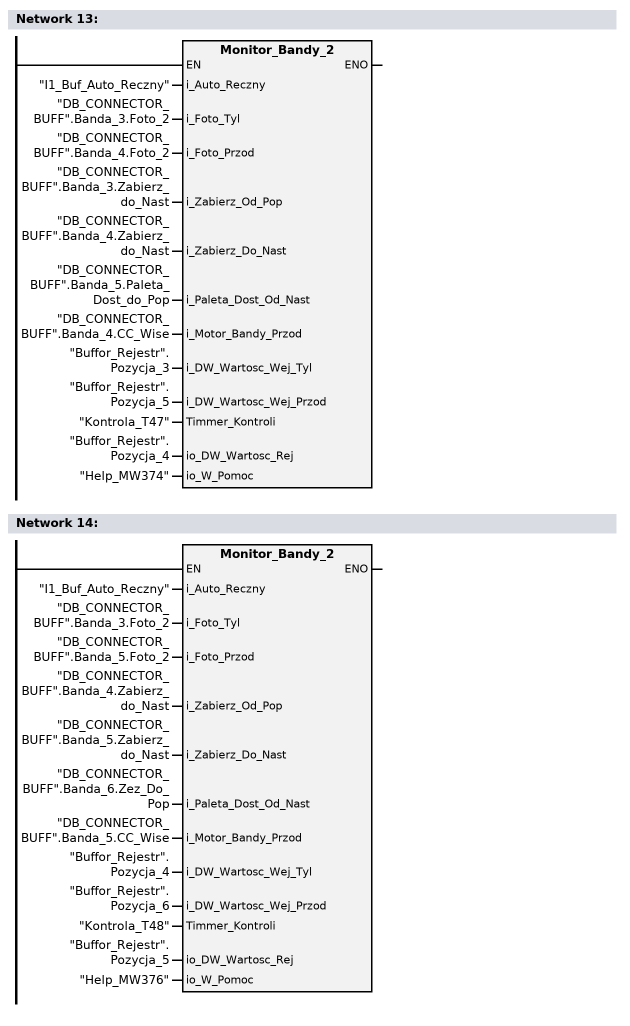
NETWORK
TITLE =
//Monitoring band 4
      CALL  "Monitor_Bandy_2" (
           i_Auto_Reczny            := "I1_Buf_Auto_Reczny",
           i_Foto_Tyl               := "DB_CONNECTOR_BUFF".Banda_3.Foto_2,
           i_Foto_Przod             := "DB_CONNECTOR_BUFF".Banda_4.Foto_2,
           i_Zabierz_Od_Pop         := "DB_CONNECTOR_BUFF".Banda_3.Zabierz_do_Nast,
           i_Zabierz_Do_Nast        := "DB_CONNECTOR_BUFF".Banda_4.Zabierz_do_Nast,
           i_Paleta_Dost_Od_Nast    := "DB_CONNECTOR_BUFF".Banda_5.Paleta_Dost_do_Pop,
           i_Motor_Bandy_Przod      := "DB_CONNECTOR_BUFF".Banda_4.CC_Wise,
           i_DW_Wartosc_Wej_Tyl     := "Buffor_Rejestr".Pozycja_3,
           i_DW_Wartosc_Wej_Przod   := "Buffor_Rejestr".Pozycja_5,
           Timmer_Kontroli          := "Kontrola_T47",
           io_DW_Wartosc_Rej        := "Buffor_Rejestr".Pozycja_4,
           io_W_Pomoc               := "Help_MW374");
NETWORK
TITLE =
//Monitoring band 5
//
      CALL  "Monitor_Bandy_2" (
           i_Auto_Reczny            := "I1_Buf_Auto_Reczny",
           i_Foto_Tyl               := "DB_CONNECTOR_BUFF".Banda_3.Foto_2,
           i_Foto_Przod             := "DB_CONNECTOR_BUFF".Banda_5.Foto_2,
           i_Zabierz_Od_Pop         := "DB_CONNECTOR_BUFF".Banda_4.Zabierz_do_Nast,
           i_Zabierz_Do_Nast        := "DB_CONNECTOR_BUFF".Banda_5.Zabierz_do_Nast,
           i_Paleta_Dost_Od_Nast    := "DB_CONNECTOR_BUFF".Banda_6.Zez_Do_Pop,
           i_Motor_Bandy_Przod      := "DB_CONNECTOR_BUFF".Banda_5.CC_Wise,
           i_DW_Wartosc_Wej_Tyl     := "Buffor_Rejestr".Pozycja_4,
           i_DW_Wartosc_Wej_Przod   := "Buffor_Rejestr".Pozycja_6,
           Timmer_Kontroli          := "Kontrola_T48",
           io_DW_Wartosc_Rej        := "Buffor_Rejestr".Pozycja_5,
           io_W_Pomoc               := "Help_MW376");
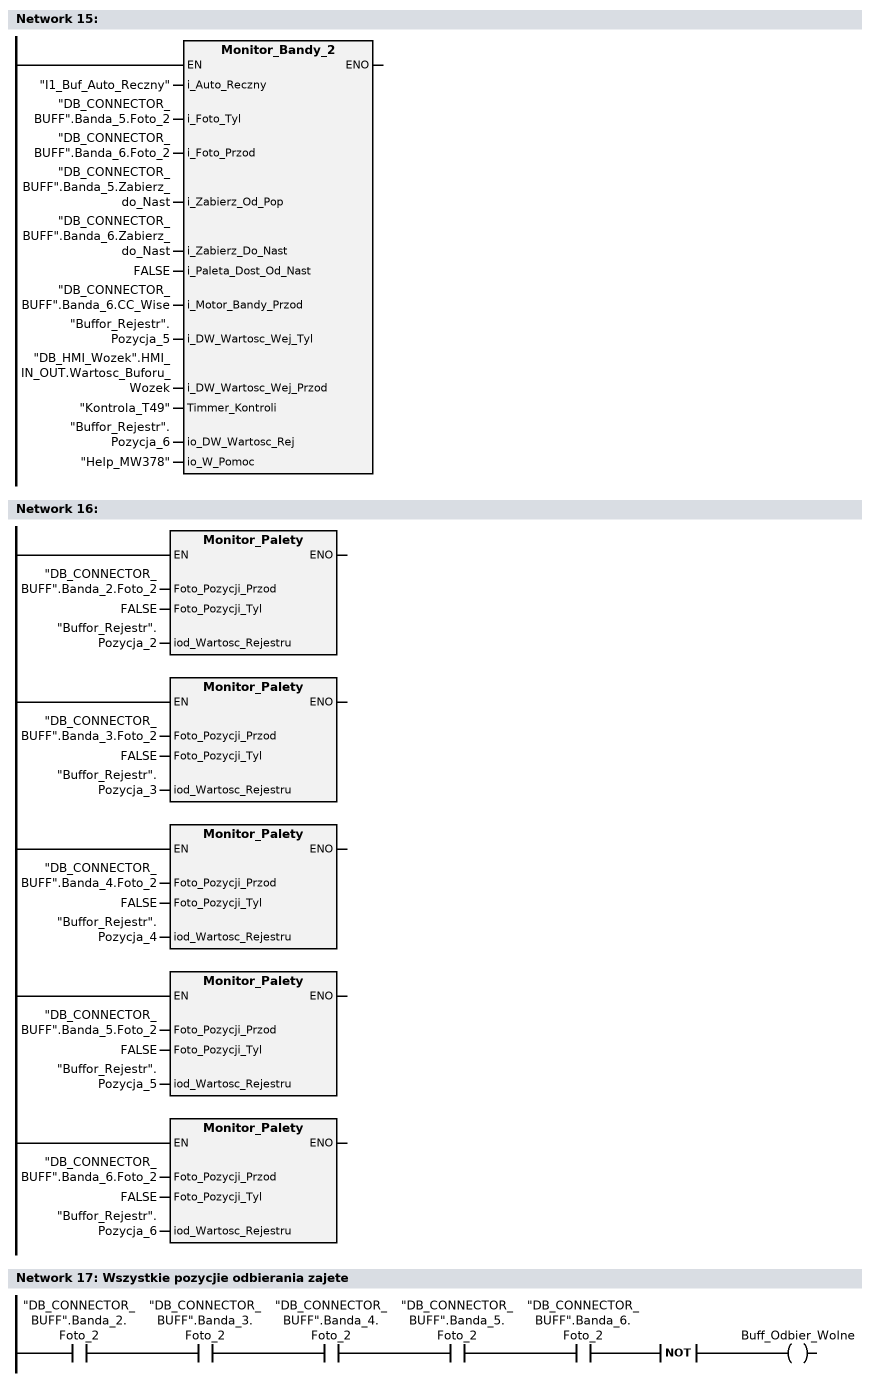
NETWORK
TITLE =
//Monitoring band 6
      CALL  "Monitor_Bandy_2" (
           i_Auto_Reczny            := "I1_Buf_Auto_Reczny",
           i_Foto_Tyl               := "DB_CONNECTOR_BUFF".Banda_5.Foto_2,
           i_Foto_Przod             := "DB_CONNECTOR_BUFF".Banda_6.Foto_2,
           i_Zabierz_Od_Pop         := "DB_CONNECTOR_BUFF".Banda_5.Zabierz_do_Nast,
           i_Zabierz_Do_Nast        := "DB_CONNECTOR_BUFF".Banda_6.Zabierz_do_Nast,
           i_Paleta_Dost_Od_Nast    := FALSE,
           i_Motor_Bandy_Przod      := "DB_CONNECTOR_BUFF".Banda_6.CC_Wise,
           i_DW_Wartosc_Wej_Tyl     := "Buffor_Rejestr".Pozycja_5,
           i_DW_Wartosc_Wej_Przod   := "DB_HMI_Wozek".HMI_IN_OUT.Wartosc_Buforu_Wozek,
           Timmer_Kontroli          := "Kontrola_T49",
           io_DW_Wartosc_Rej        := "Buffor_Rejestr".Pozycja_6,
           io_W_Pomoc               := "Help_MW378");
NETWORK
TITLE =
//Zaznaczenie czy jest paleta
      CALL  "Monitor_Palety" (
           Foto_Pozycji_Przod       := "DB_CONNECTOR_BUFF".Banda_2.Foto_2,
           Foto_Pozycji_Tyl         := FALSE,
           iod_Wartosc_Rejestru     := "Buffor_Rejestr".Pozycja_2);
      CALL  "Monitor_Palety" (
           Foto_Pozycji_Przod       := "DB_CONNECTOR_BUFF".Banda_3.Foto_2,
           Foto_Pozycji_Tyl         := FALSE,
           iod_Wartosc_Rejestru     := "Buffor_Rejestr".Pozycja_3);
      CALL  "Monitor_Palety" (
           Foto_Pozycji_Przod       := "DB_CONNECTOR_BUFF".Banda_4.Foto_2,
           Foto_Pozycji_Tyl         := FALSE,
           iod_Wartosc_Rejestru     := "Buffor_Rejestr".Pozycja_4);
      CALL  "Monitor_Palety" (
           Foto_Pozycji_Przod       := "DB_CONNECTOR_BUFF".Banda_5.Foto_2,
           Foto_Pozycji_Tyl         := FALSE,
           iod_Wartosc_Rejestru     := "Buffor_Rejestr".Pozycja_5);
      CALL  "Monitor_Palety" (
           Foto_Pozycji_Przod       := "DB_CONNECTOR_BUFF".Banda_6.Foto_2,
           Foto_Pozycji_Tyl         := FALSE,
           iod_Wartosc_Rejestru     := "Buffor_Rejestr".Pozycja_6);
NETWORK
TITLE = Wszystkie pozycjie odbierania zajete
//Sprawdzenie czy wszystkie pozycje sa zajete
      A     "DB_CONNECTOR_BUFF".Banda_2.Foto_2;
      A     "DB_CONNECTOR_BUFF".Banda_3.Foto_2;
      A     "DB_CONNECTOR_BUFF".Banda_4.Foto_2;
      A     "DB_CONNECTOR_BUFF".Banda_5.Foto_2;
      A     "DB_CONNECTOR_BUFF".Banda_6.Foto_2;
      NOT;
      =     "Buff_Odbier_Wolne";
END_FUNCTION_BLOCK

FUNCTION_BLOCK "Stan_Intro_Pob_I1"	// FB 7
//Stanowisko intro Pobieranie
//Linia zlozona z 5 band odbierajacych
//
//
//BW B16 B15 B14 B13 B12 
//             <===
//
//5 band kierunek zanegowany
VERSION : 0.1
VAR
  Banda_12 : FB 33;
  Banda_13 : FB 33;
  Banda_14 : FB 33;
  Banda_15 : FB 33;
  Banda_16 : FB 33;
END_VAR
VAR_TEMP
  Help_Bit_1 : BOOL ;
  Help_Reczny_Przod : BOOL ;
  Help_Reczny_Tyl : BOOL ;
  Help_int : INT ;
  Help_Dword : DWORD ;
  Help_INT_1 : DINT ;
END_VAR
BEGIN
NETWORK
TITLE =
//Ten Network celowo jest wolny
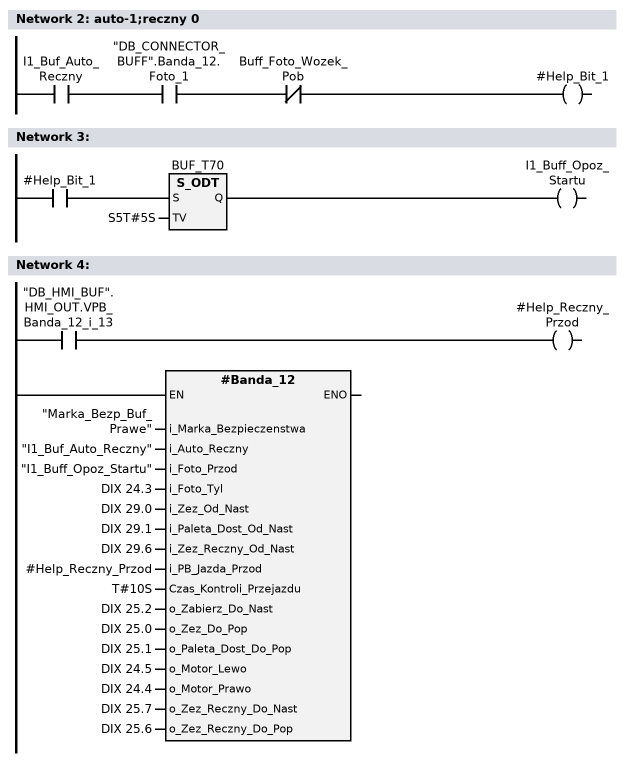
NETWORK
TITLE = auto-1;reczny 0
      A     "I1_Buf_Auto_Reczny";
      A     "DB_CONNECTOR_BUFF".Banda_12.Foto_1;
      AN    "Buff_Foto_Wozek_Pob";
      =     #Help_Bit_1;
NETWORK
TITLE =
//Opoznienie startu po polozeniu palety
//
      A     #Help_Bit_1;
      L     S5T#5S;
      SD    "BUF_T70";
      NOP   0;
      NOP   0;
      NOP   0;
      A     "BUF_T70";
      =     "I1_Buff_Opoz_Startu";
NETWORK
TITLE =
//Banda 12
      O     "DB_HMI_BUF".HMI_OUT.VPB_Banda_12_i_13;
      =     #Help_Reczny_Przod;
      CALL  #Banda_12 (
           i_Marka_Bezpieczenstwa   := "Marka_Bezp_Buf_Prawe",
           i_Auto_Reczny            := "I1_Buf_Auto_Reczny",
           i_Foto_Przod             := "I1_Buff_Opoz_Startu",
           i_Foto_Tyl               := DIX 24.3,
           i_Zez_Od_Nast            := DIX 29.0,
           i_Paleta_Dost_Od_Nast    := DIX 29.1,
           i_Zez_Reczny_Od_Nast     := DIX 29.6,
           i_PB_Jazda_Przod         := #Help_Reczny_Przod,
           Czas_Kontroli_Przejazdu  := T#10S,
           o_Zabierz_Do_Nast        := DIX 25.2,
           o_Zez_Do_Pop             := DIX 25.0,
           o_Paleta_Dost_Do_Pop     := DIX 25.1,
           o_Motor_Lewo             := DIX 24.5,
           o_Motor_Prawo            := DIX 24.4,
           o_Zez_Reczny_Do_Nast     := DIX 25.7,
           o_Zez_Reczny_Do_Pop      := DIX 25.6);
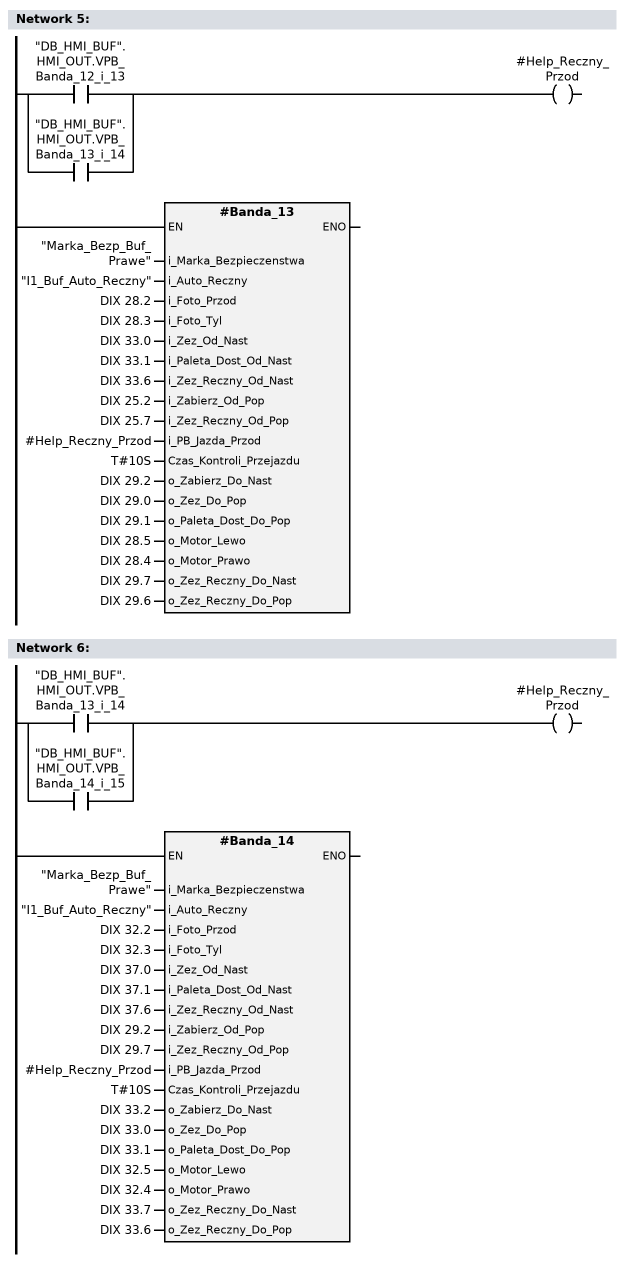
NETWORK
TITLE =
//Banda 13
      O     "DB_HMI_BUF".HMI_OUT.VPB_Banda_12_i_13;
      O     "DB_HMI_BUF".HMI_OUT.VPB_Banda_13_i_14;
      =     #Help_Reczny_Przod;
      CALL  #Banda_13 (
           i_Marka_Bezpieczenstwa   := "Marka_Bezp_Buf_Prawe",
           i_Auto_Reczny            := "I1_Buf_Auto_Reczny",
           i_Foto_Przod             := DIX 28.2,
           i_Foto_Tyl               := DIX 28.3,
           i_Zez_Od_Nast            := DIX 33.0,
           i_Paleta_Dost_Od_Nast    := DIX 33.1,
           i_Zez_Reczny_Od_Nast     := DIX 33.6,
           i_Zabierz_Od_Pop         := DIX 25.2,
           i_Zez_Reczny_Od_Pop      := DIX 25.7,
           i_PB_Jazda_Przod         := #Help_Reczny_Przod,
           Czas_Kontroli_Przejazdu  := T#10S,
           o_Zabierz_Do_Nast        := DIX 29.2,
           o_Zez_Do_Pop             := DIX 29.0,
           o_Paleta_Dost_Do_Pop     := DIX 29.1,
           o_Motor_Lewo             := DIX 28.5,
           o_Motor_Prawo            := DIX 28.4,
           o_Zez_Reczny_Do_Nast     := DIX 29.7,
           o_Zez_Reczny_Do_Pop      := DIX 29.6);
NETWORK
TITLE =
//Banda 14
      O     "DB_HMI_BUF".HMI_OUT.VPB_Banda_13_i_14;
      O     "DB_HMI_BUF".HMI_OUT.VPB_Banda_14_i_15;
      =     #Help_Reczny_Przod;
      CALL  #Banda_14 (
           i_Marka_Bezpieczenstwa   := "Marka_Bezp_Buf_Prawe",
           i_Auto_Reczny            := "I1_Buf_Auto_Reczny",
           i_Foto_Przod             := DIX 32.2,
           i_Foto_Tyl               := DIX 32.3,
           i_Zez_Od_Nast            := DIX 37.0,
           i_Paleta_Dost_Od_Nast    := DIX 37.1,
           i_Zez_Reczny_Od_Nast     := DIX 37.6,
           i_Zabierz_Od_Pop         := DIX 29.2,
           i_Zez_Reczny_Od_Pop      := DIX 29.7,
           i_PB_Jazda_Przod         := #Help_Reczny_Przod,
           Czas_Kontroli_Przejazdu  := T#10S,
           o_Zabierz_Do_Nast        := DIX 33.2,
           o_Zez_Do_Pop             := DIX 33.0,
           o_Paleta_Dost_Do_Pop     := DIX 33.1,
           o_Motor_Lewo             := DIX 32.5,
           o_Motor_Prawo            := DIX 32.4,
           o_Zez_Reczny_Do_Nast     := DIX 33.7,
           o_Zez_Reczny_Do_Pop      := DIX 33.6);
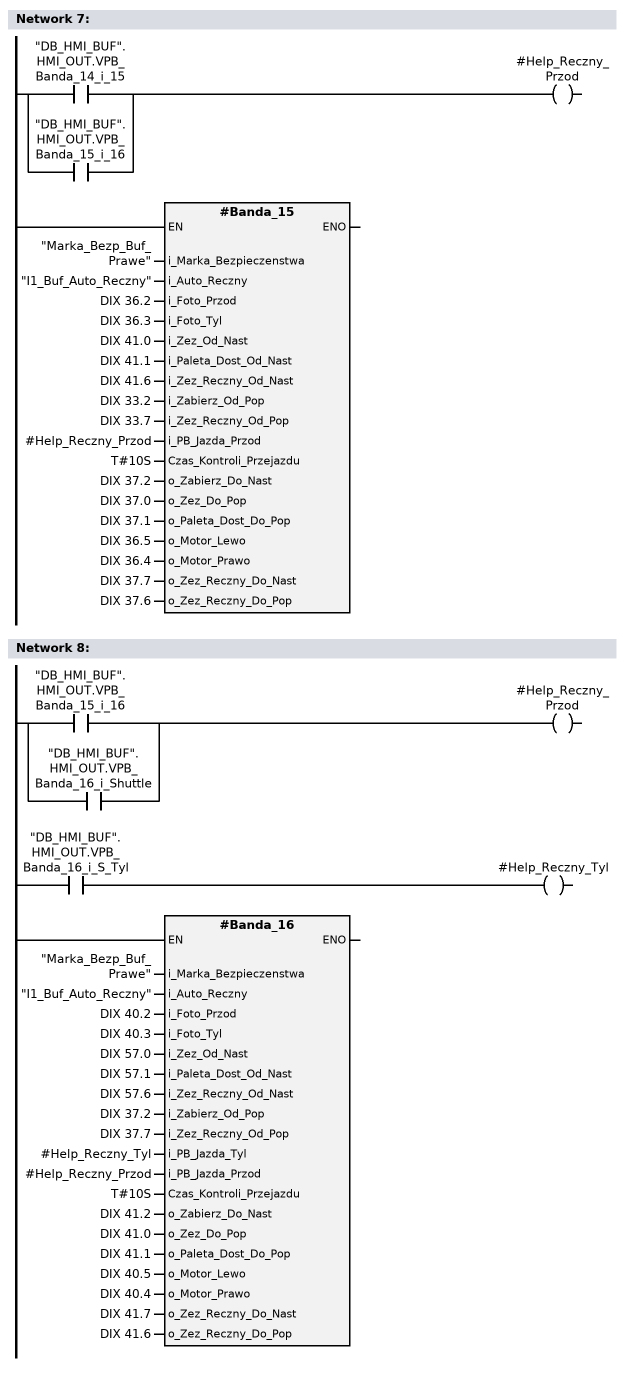
NETWORK
TITLE =
//Banda 15
      O     "DB_HMI_BUF".HMI_OUT.VPB_Banda_14_i_15;
      O     "DB_HMI_BUF".HMI_OUT.VPB_Banda_15_i_16;
      =     #Help_Reczny_Przod;
      CALL  #Banda_15 (
           i_Marka_Bezpieczenstwa   := "Marka_Bezp_Buf_Prawe",
           i_Auto_Reczny            := "I1_Buf_Auto_Reczny",
           i_Foto_Przod             := DIX 36.2,
           i_Foto_Tyl               := DIX 36.3,
           i_Zez_Od_Nast            := DIX 41.0,
           i_Paleta_Dost_Od_Nast    := DIX 41.1,
           i_Zez_Reczny_Od_Nast     := DIX 41.6,
           i_Zabierz_Od_Pop         := DIX 33.2,
           i_Zez_Reczny_Od_Pop      := DIX 33.7,
           i_PB_Jazda_Przod         := #Help_Reczny_Przod,
           Czas_Kontroli_Przejazdu  := T#10S,
           o_Zabierz_Do_Nast        := DIX 37.2,
           o_Zez_Do_Pop             := DIX 37.0,
           o_Paleta_Dost_Do_Pop     := DIX 37.1,
           o_Motor_Lewo             := DIX 36.5,
           o_Motor_Prawo            := DIX 36.4,
           o_Zez_Reczny_Do_Nast     := DIX 37.7,
           o_Zez_Reczny_Do_Pop      := DIX 37.6);
NETWORK
TITLE =
//Banda 16
      O     "DB_HMI_BUF".HMI_OUT.VPB_Banda_15_i_16;
      O     "DB_HMI_BUF".HMI_OUT.VPB_Banda_16_i_Shuttle;
      =     #Help_Reczny_Przod;
      O     "DB_HMI_BUF".HMI_OUT.VPB_Banda_16_i_S_Tyl;
      =     #Help_Reczny_Tyl;
      CALL  #Banda_16 (
           i_Marka_Bezpieczenstwa   := "Marka_Bezp_Buf_Prawe",
           i_Auto_Reczny            := "I1_Buf_Auto_Reczny",
           i_Foto_Przod             := DIX 40.2,
           i_Foto_Tyl               := DIX 40.3,
           i_Zez_Od_Nast            := DIX 57.0,
           i_Paleta_Dost_Od_Nast    := DIX 57.1,
           i_Zez_Reczny_Od_Nast     := DIX 57.6,
           i_Zabierz_Od_Pop         := DIX 37.2,
           i_Zez_Reczny_Od_Pop      := DIX 37.7,
           i_PB_Jazda_Tyl           := #Help_Reczny_Tyl,
           i_PB_Jazda_Przod         := #Help_Reczny_Przod,
           Czas_Kontroli_Przejazdu  := T#10S,
           o_Zabierz_Do_Nast        := DIX 41.2,
           o_Zez_Do_Pop             := DIX 41.0,
           o_Paleta_Dost_Do_Pop     := DIX 41.1,
           o_Motor_Lewo             := DIX 40.5,
           o_Motor_Prawo            := DIX 40.4,
           o_Zez_Reczny_Do_Nast     := DIX 41.7,
           o_Zez_Reczny_Do_Pop      := DIX 41.6);
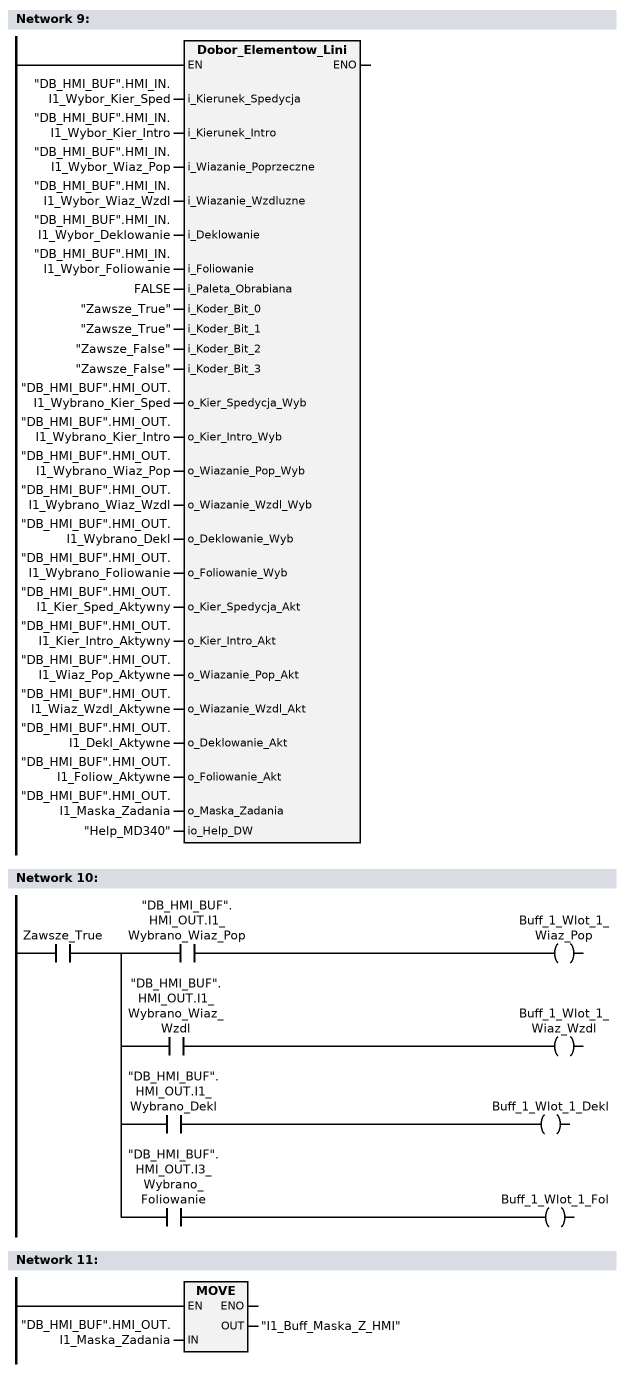
NETWORK
TITLE =
//Wybor Elementow na lini
      CALL  "Dobor_Elementow_Lini" (
           i_Kierunek_Spedycja      := "DB_HMI_BUF".HMI_IN.I1_Wybor_Kier_Sped,
           i_Kierunek_Intro         := "DB_HMI_BUF".HMI_IN.I1_Wybor_Kier_Intro,
           i_Wiazanie_Poprzeczne    := "DB_HMI_BUF".HMI_IN.I1_Wybor_Wiaz_Pop,
           i_Wiazanie_Wzdluzne      := "DB_HMI_BUF".HMI_IN.I1_Wybor_Wiaz_Wzdl,
           i_Deklowanie             := "DB_HMI_BUF".HMI_IN.I1_Wybor_Deklowanie,
           i_Foliowanie             := "DB_HMI_BUF".HMI_IN.I1_Wybor_Foliowanie,
           i_Paleta_Obrabiana       := FALSE,
           i_Koder_Bit_0            := "Zawsze_True",
           i_Koder_Bit_1            := "Zawsze_True",
           i_Koder_Bit_2            := "Zawsze_False",
           i_Koder_Bit_3            := "Zawsze_False",
           o_Kier_Spedycja_Wyb      := "DB_HMI_BUF".HMI_OUT.I1_Wybrano_Kier_Sped,
           o_Kier_Intro_Wyb         := "DB_HMI_BUF".HMI_OUT.I1_Wybrano_Kier_Intro,
           o_Wiazanie_Pop_Wyb       := "DB_HMI_BUF".HMI_OUT.I1_Wybrano_Wiaz_Pop,
           o_Wiazanie_Wzdl_Wyb      := "DB_HMI_BUF".HMI_OUT.I1_Wybrano_Wiaz_Wzdl,
           o_Deklowanie_Wyb         := "DB_HMI_BUF".HMI_OUT.I1_Wybrano_Dekl,
           o_Foliowanie_Wyb         := "DB_HMI_BUF".HMI_OUT.I1_Wybrano_Foliowanie,
           o_Kier_Spedycja_Akt      := "DB_HMI_BUF".HMI_OUT.I1_Kier_Sped_Aktywny,
           o_Kier_Intro_Akt         := "DB_HMI_BUF".HMI_OUT.I1_Kier_Intro_Aktywny,
           o_Wiazanie_Pop_Akt       := "DB_HMI_BUF".HMI_OUT.I1_Wiaz_Pop_Aktywne,
           o_Wiazanie_Wzdl_Akt      := "DB_HMI_BUF".HMI_OUT.I1_Wiaz_Wzdl_Aktywne,
           o_Deklowanie_Akt         := "DB_HMI_BUF".HMI_OUT.I1_Dekl_Aktywne,
           o_Foliowanie_Akt         := "DB_HMI_BUF".HMI_OUT.I1_Foliow_Aktywne,
           o_Maska_Zadania          := "DB_HMI_BUF".HMI_OUT.I1_Maska_Zadania,
           io_Help_DW               := "Help_MD340");
NETWORK
TITLE =
//Wyswietlenie lampek zadania lini
      A     "Zawsze_True";
      =     L 12.0;
      A     L 12.0;
      A     "DB_HMI_BUF".HMI_OUT.I1_Wybrano_Wiaz_Pop;
      =     "Buff_1_Wlot_1_Wiaz_Pop";
      A     L 12.0;
      A     "DB_HMI_BUF".HMI_OUT.I1_Wybrano_Wiaz_Wzdl;
      =     "Buff_1_Wlot_1_Wiaz_Wzdl";
      A     L 12.0;
      A     "DB_HMI_BUF".HMI_OUT.I1_Wybrano_Dekl;
      =     "Buff_1_Wlot_1_Dekl";
      A     L 12.0;
      A     "DB_HMI_BUF".HMI_OUT.I3_Wybrano_Foliowanie;
      =     "Buff_1_Wlot_1_Fol";
NETWORK
TITLE =
//Przypisanie maski zadania do bandy wejsciowej
      L     "DB_HMI_BUF".HMI_OUT.I1_Maska_Zadania;
      T     "I1_Buff_Maska_Z_HMI";
      NOP   0;
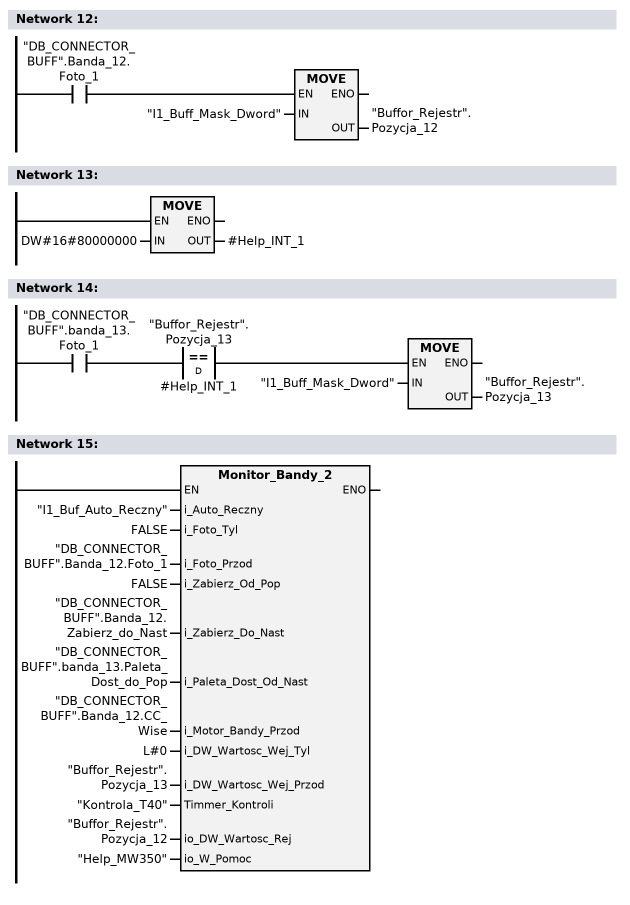
NETWORK
TITLE =
//Zbudowanie z maski podwojnego slowa
      A     "DB_CONNECTOR_BUFF".Banda_12.Foto_1;
      JNB   _001;
      L     "I1_Buff_Mask_Dword";
      T     "Buffor_Rejestr".Pozycja_12;
_001: NOP   0;
NETWORK
TITLE =
      L     DW#16#80000000;
      T     #Help_INT_1;
      NOP   0;
NETWORK
TITLE =
//sprawdzenie dla fotokomorki bandy 13
      A     "DB_CONNECTOR_BUFF".banda_13.Foto_1;
      A(;
      L     "Buffor_Rejestr".Pozycja_13;
      L     #Help_INT_1;
      ==D;
      );
      JNB   _002;
      L     "I1_Buff_Mask_Dword";
      T     "Buffor_Rejestr".Pozycja_13;
_002: NOP   0;
NETWORK
TITLE =
//Monitoring band 12
      CALL  "Monitor_Bandy_2" (
           i_Auto_Reczny            := "I1_Buf_Auto_Reczny",
           i_Foto_Tyl               := FALSE,
           i_Foto_Przod             := "DB_CONNECTOR_BUFF".Banda_12.Foto_1,
           i_Zabierz_Od_Pop         := FALSE,
           i_Zabierz_Do_Nast        := "DB_CONNECTOR_BUFF".Banda_12.Zabierz_do_Nast,
           i_Paleta_Dost_Od_Nast    := "DB_CONNECTOR_BUFF".banda_13.Paleta_Dost_do_Pop,
           i_Motor_Bandy_Przod      := "DB_CONNECTOR_BUFF".Banda_12.CC_Wise,
           i_DW_Wartosc_Wej_Tyl     := L#0,
           i_DW_Wartosc_Wej_Przod   := "Buffor_Rejestr".Pozycja_13,
           Timmer_Kontroli          := "Kontrola_T40",
           io_DW_Wartosc_Rej        := "Buffor_Rejestr".Pozycja_12,
           io_W_Pomoc               := "Help_MW350");
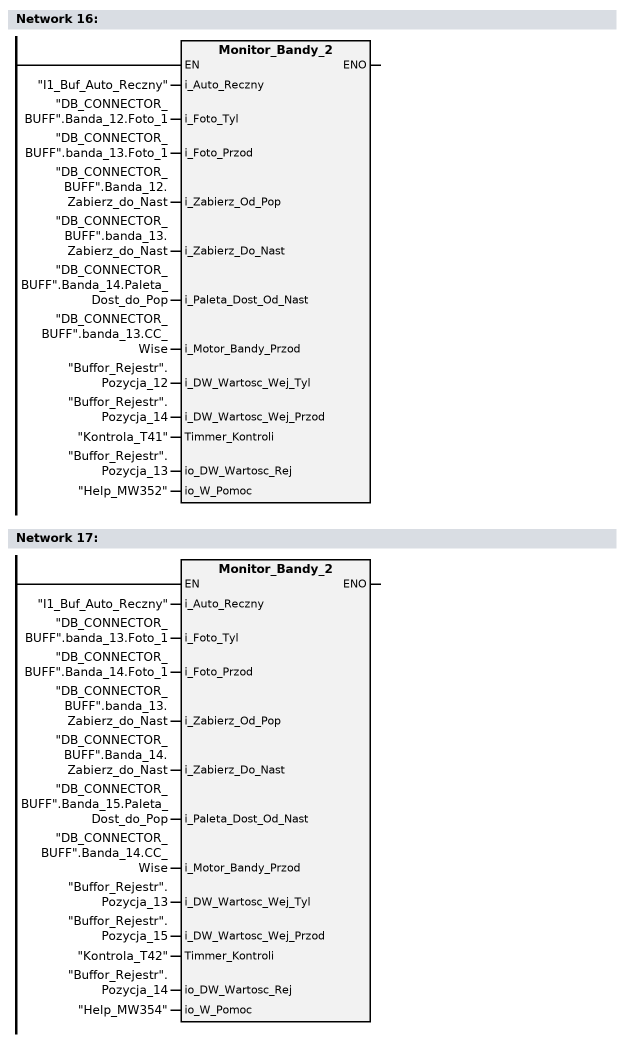
NETWORK
TITLE =
//Monitoring band 13
      CALL  "Monitor_Bandy_2" (
           i_Auto_Reczny            := "I1_Buf_Auto_Reczny",
           i_Foto_Tyl               := "DB_CONNECTOR_BUFF".Banda_12.Foto_1,
           i_Foto_Przod             := "DB_CONNECTOR_BUFF".banda_13.Foto_1,
           i_Zabierz_Od_Pop         := "DB_CONNECTOR_BUFF".Banda_12.Zabierz_do_Nast,
           i_Zabierz_Do_Nast        := "DB_CONNECTOR_BUFF".banda_13.Zabierz_do_Nast,
           i_Paleta_Dost_Od_Nast    := "DB_CONNECTOR_BUFF".Banda_14.Paleta_Dost_do_Pop,
           i_Motor_Bandy_Przod      := "DB_CONNECTOR_BUFF".banda_13.CC_Wise,
           i_DW_Wartosc_Wej_Tyl     := "Buffor_Rejestr".Pozycja_12,
           i_DW_Wartosc_Wej_Przod   := "Buffor_Rejestr".Pozycja_14,
           Timmer_Kontroli          := "Kontrola_T41",
           io_DW_Wartosc_Rej        := "Buffor_Rejestr".Pozycja_13,
           io_W_Pomoc               := "Help_MW352");
NETWORK
TITLE =
//Monitoring band 14
      CALL  "Monitor_Bandy_2" (
           i_Auto_Reczny            := "I1_Buf_Auto_Reczny",
           i_Foto_Tyl               := "DB_CONNECTOR_BUFF".banda_13.Foto_1,
           i_Foto_Przod             := "DB_CONNECTOR_BUFF".Banda_14.Foto_1,
           i_Zabierz_Od_Pop         := "DB_CONNECTOR_BUFF".banda_13.Zabierz_do_Nast,
           i_Zabierz_Do_Nast        := "DB_CONNECTOR_BUFF".Banda_14.Zabierz_do_Nast,
           i_Paleta_Dost_Od_Nast    := "DB_CONNECTOR_BUFF".Banda_15.Paleta_Dost_do_Pop,
           i_Motor_Bandy_Przod      := "DB_CONNECTOR_BUFF".Banda_14.CC_Wise,
           i_DW_Wartosc_Wej_Tyl     := "Buffor_Rejestr".Pozycja_13,
           i_DW_Wartosc_Wej_Przod   := "Buffor_Rejestr".Pozycja_15,
           Timmer_Kontroli          := "Kontrola_T42",
           io_DW_Wartosc_Rej        := "Buffor_Rejestr".Pozycja_14,
           io_W_Pomoc               := "Help_MW354");
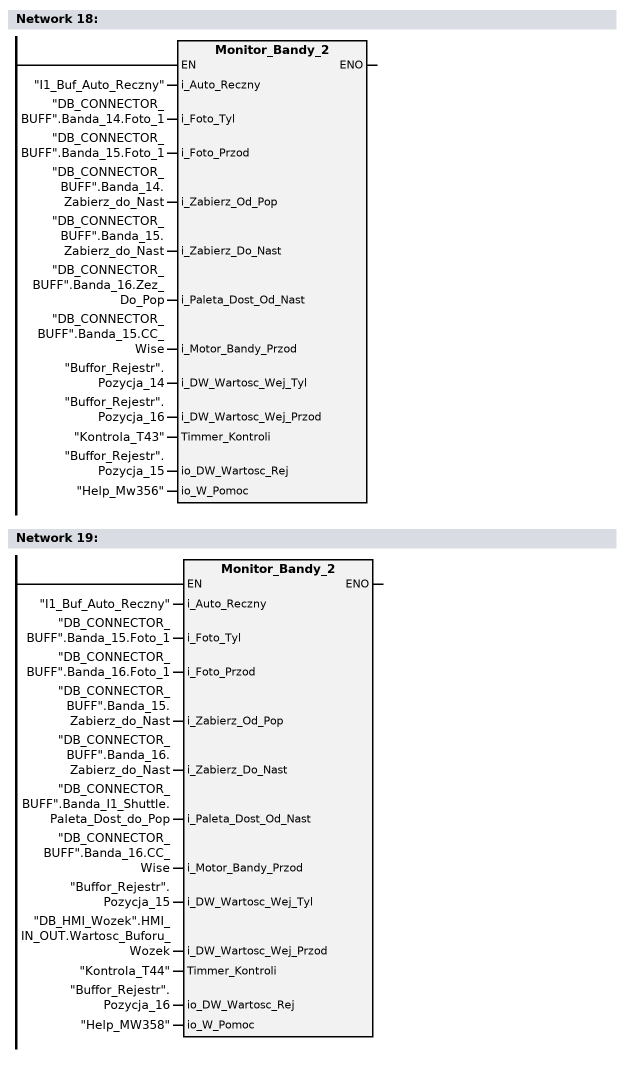
NETWORK
TITLE =
//Monitoring band 15
//
      CALL  "Monitor_Bandy_2" (
           i_Auto_Reczny            := "I1_Buf_Auto_Reczny",
           i_Foto_Tyl               := "DB_CONNECTOR_BUFF".Banda_14.Foto_1,
           i_Foto_Przod             := "DB_CONNECTOR_BUFF".Banda_15.Foto_1,
           i_Zabierz_Od_Pop         := "DB_CONNECTOR_BUFF".Banda_14.Zabierz_do_Nast,
           i_Zabierz_Do_Nast        := "DB_CONNECTOR_BUFF".Banda_15.Zabierz_do_Nast,
           i_Paleta_Dost_Od_Nast    := "DB_CONNECTOR_BUFF".Banda_16.Zez_Do_Pop,
           i_Motor_Bandy_Przod      := "DB_CONNECTOR_BUFF".Banda_15.CC_Wise,
           i_DW_Wartosc_Wej_Tyl     := "Buffor_Rejestr".Pozycja_14,
           i_DW_Wartosc_Wej_Przod   := "Buffor_Rejestr".Pozycja_16,
           Timmer_Kontroli          := "Kontrola_T43",
           io_DW_Wartosc_Rej        := "Buffor_Rejestr".Pozycja_15,
           io_W_Pomoc               := "Help_Mw356");
NETWORK
TITLE =
//Monitoring band 16
      CALL  "Monitor_Bandy_2" (
           i_Auto_Reczny            := "I1_Buf_Auto_Reczny",
           i_Foto_Tyl               := "DB_CONNECTOR_BUFF".Banda_15.Foto_1,
           i_Foto_Przod             := "DB_CONNECTOR_BUFF".Banda_16.Foto_1,
           i_Zabierz_Od_Pop         := "DB_CONNECTOR_BUFF".Banda_15.Zabierz_do_Nast,
           i_Zabierz_Do_Nast        := "DB_CONNECTOR_BUFF".Banda_16.Zabierz_do_Nast,
           i_Paleta_Dost_Od_Nast    := "DB_CONNECTOR_BUFF".Banda_I1_Shuttle.Paleta_Dost_do_Pop,
           i_Motor_Bandy_Przod      := "DB_CONNECTOR_BUFF".Banda_16.CC_Wise,
           i_DW_Wartosc_Wej_Tyl     := "Buffor_Rejestr".Pozycja_15,
           i_DW_Wartosc_Wej_Przod   := "DB_HMI_Wozek".HMI_IN_OUT.Wartosc_Buforu_Wozek,
           Timmer_Kontroli          := "Kontrola_T44",
           io_DW_Wartosc_Rej        := "Buffor_Rejestr".Pozycja_16,
           io_W_Pomoc               := "Help_MW358");
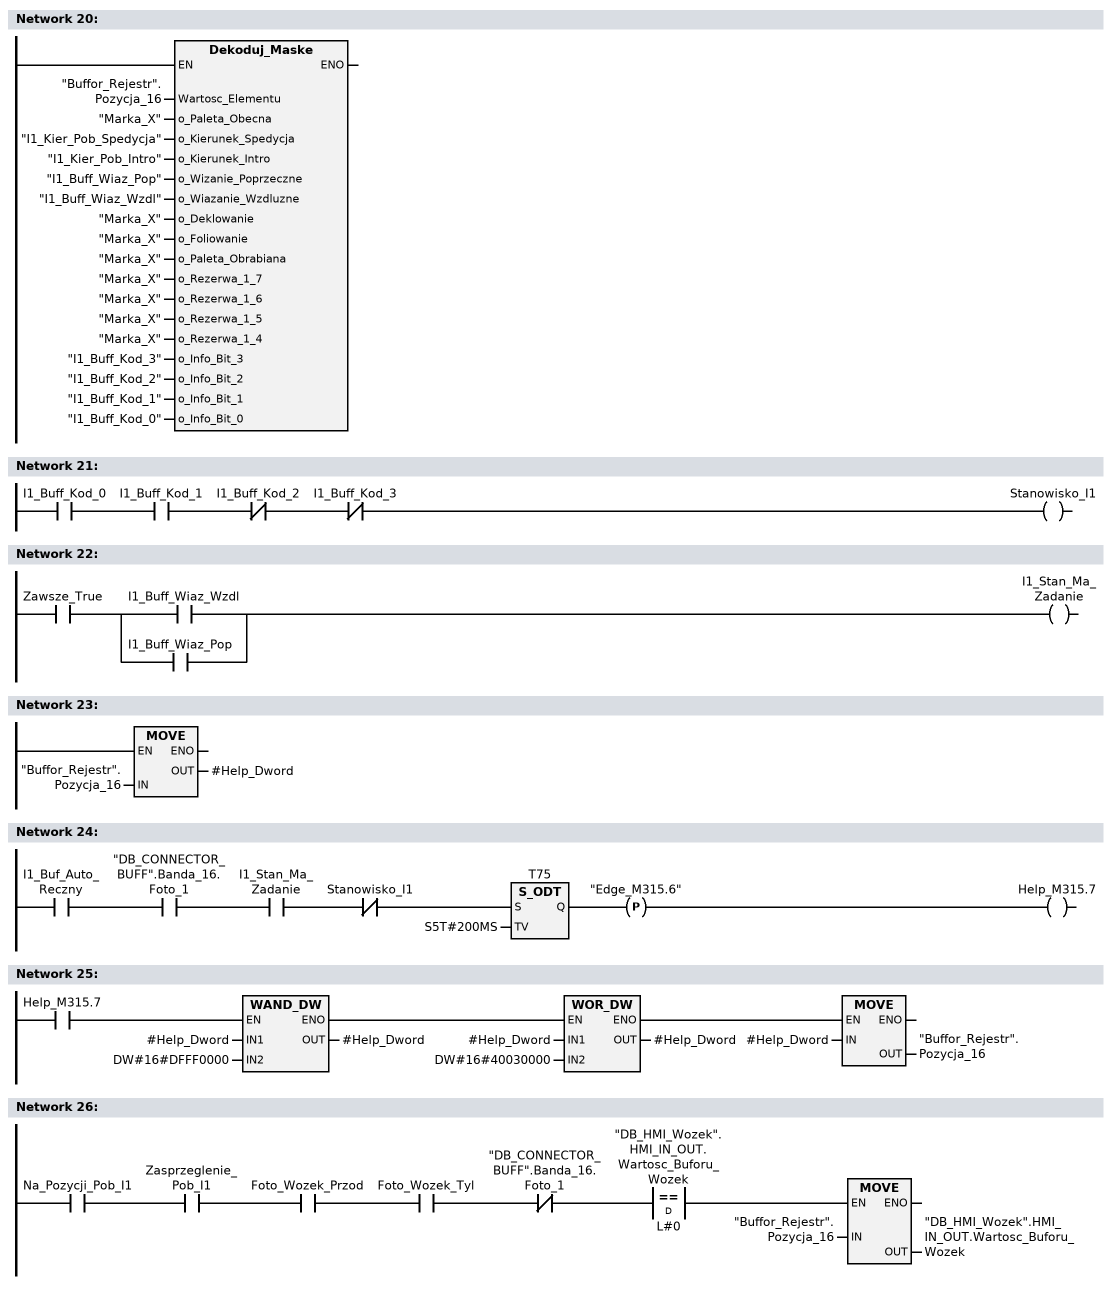
NETWORK
TITLE =
//Dekouj maske
//Potrzebne do okreslenia kierunku kursu
      CALL  "Dekoduj_Maske" (
           Wartosc_Elementu         := "Buffor_Rejestr".Pozycja_16,
           o_Paleta_Obecna          := "Marka_X",
           o_Kierunek_Spedycja      := "I1_Kier_Pob_Spedycja",
           o_Kierunek_Intro         := "I1_Kier_Pob_Intro",
           o_Wizanie_Poprzeczne     := "I1_Buff_Wiaz_Pop",
           o_Wiazanie_Wzdluzne      := "I1_Buff_Wiaz_Wzdl",
           o_Deklowanie             := "Marka_X",
           o_Foliowanie             := "Marka_X",
           o_Paleta_Obrabiana       := "Marka_X",
           o_Rezerwa_1_7            := "Marka_X",
           o_Rezerwa_1_6            := "Marka_X",
           o_Rezerwa_1_5            := "Marka_X",
           o_Rezerwa_1_4            := "Marka_X",
           o_Info_Bit_3             := "I1_Buff_Kod_3",
           o_Info_Bit_2             := "I1_Buff_Kod_2",
           o_Info_Bit_1             := "I1_Buff_Kod_1",
           o_Info_Bit_0             := "I1_Buff_Kod_0");
NETWORK
TITLE =
//Stanowisko intro
      A     "I1_Buff_Kod_0";
      A     "I1_Buff_Kod_1";
      AN    "I1_Buff_Kod_2";
      AN    "I1_Buff_Kod_3";
      =     "Stanowisko_I1";
NETWORK
TITLE =
//Stanowisko intro ma jakies zadanie
      A     "Zawsze_True";
      A(;
      O     "I1_Buff_Wiaz_Wzdl";
      O     "I1_Buff_Wiaz_Pop";
      );
      =     "I1_Stan_Ma_Zadanie";
NETWORK
TITLE =
      L     "Buffor_Rejestr".Pozycja_16;
      T     #Help_Dword;
      NOP   0;
NETWORK
TITLE =
//Przepisanie wartosci nowej wartosci kodu jesli jest zadanie a paleta nie znana
//Domyslnie wysylana jest na Gender
      A(;
      A     "I1_Buf_Auto_Reczny";
      A     "DB_CONNECTOR_BUFF".Banda_16.Foto_1;
      A     "I1_Stan_Ma_Zadanie";
      AN    "Stanowisko_I1";
      L     S5T#200MS;
      SD    "T75";
      NOP   0;
      NOP   0;
      NOP   0;
      A     "T75";
      );
      FP    "Edge_M315.6";
      =     "Help_M315.7";
NETWORK
TITLE =
//Przypisanie nowej wartosci do palety
      A(;
      A(;
      A     "Help_M315.7";
      JNB   _003;
      L     #Help_Dword;
      L     DW#16#DFFF0000;
      AD;
      T     #Help_Dword;
      SET;
      SAVE;
      CLR;
_003: A     BR;
      );
      JNB   _004;
      L     #Help_Dword;
      L     DW#16#40030000;
      OD;
      T     #Help_Dword;
      SET;
      SAVE;
      CLR;
_004: A     BR;
      );
      JNB   _005;
      L     #Help_Dword;
      T     "Buffor_Rejestr".Pozycja_16;
_005: NOP   0;
NETWORK
TITLE =
//db128.db208 -wartosc rejestru na wozka
      A     "Na_Pozycji_Pob_I1";
      A     "Zasprzeglenie_Pob_I1";
      A     "Foto_Wozek_Przod";
      A     "Foto_Wozek_Tyl";
      AN    "DB_CONNECTOR_BUFF".Banda_16.Foto_1;
      A(;
      L     "DB_HMI_Wozek".HMI_IN_OUT.Wartosc_Buforu_Wozek;
      L     L#0;
      ==D;
      );
      JNB   _006;
      L     "Buffor_Rejestr".Pozycja_16;
      T     "DB_HMI_Wozek".HMI_IN_OUT.Wartosc_Buforu_Wozek;
_006: NOP   0;
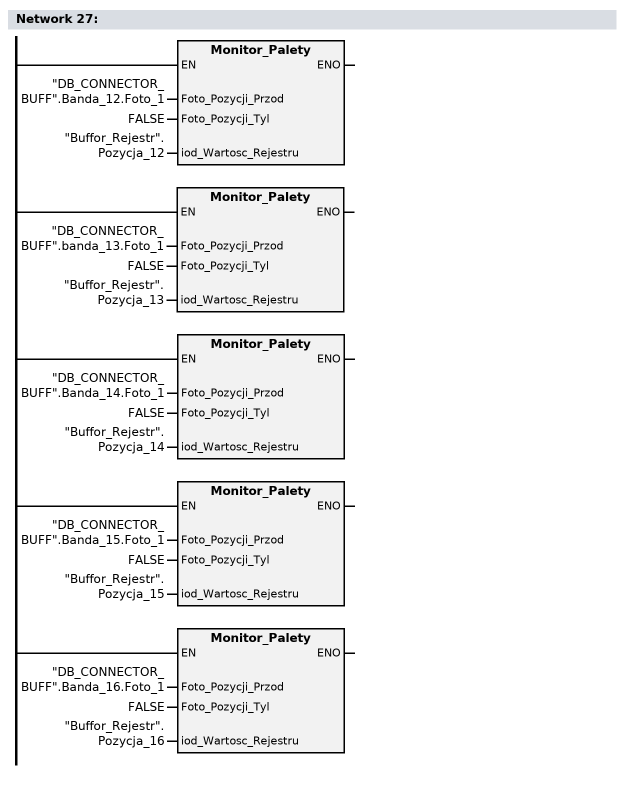
NETWORK
TITLE =
//Monitor palet
      CALL  "Monitor_Palety" (
           Foto_Pozycji_Przod       := "DB_CONNECTOR_BUFF".Banda_12.Foto_1,
           Foto_Pozycji_Tyl         := FALSE,
           iod_Wartosc_Rejestru     := "Buffor_Rejestr".Pozycja_12);
      CALL  "Monitor_Palety" (
           Foto_Pozycji_Przod       := "DB_CONNECTOR_BUFF".banda_13.Foto_1,
           Foto_Pozycji_Tyl         := FALSE,
           iod_Wartosc_Rejestru     := "Buffor_Rejestr".Pozycja_13);
      CALL  "Monitor_Palety" (
           Foto_Pozycji_Przod       := "DB_CONNECTOR_BUFF".Banda_14.Foto_1,
           Foto_Pozycji_Tyl         := FALSE,
           iod_Wartosc_Rejestru     := "Buffor_Rejestr".Pozycja_14);
      CALL  "Monitor_Palety" (
           Foto_Pozycji_Przod       := "DB_CONNECTOR_BUFF".Banda_15.Foto_1,
           Foto_Pozycji_Tyl         := FALSE,
           iod_Wartosc_Rejestru     := "Buffor_Rejestr".Pozycja_15);
      CALL  "Monitor_Palety" (
           Foto_Pozycji_Przod       := "DB_CONNECTOR_BUFF".Banda_16.Foto_1,
           Foto_Pozycji_Tyl         := FALSE,
           iod_Wartosc_Rejestru     := "Buffor_Rejestr".Pozycja_16);
END_FUNCTION_BLOCK

FUNCTION_BLOCK "Stan_Intro_Pob_I2"	// FB 8
//Stanowisko intro Pobieranie
//Linia zlozona z 5 band odbierajacych
//
//
//B7 B8 BW
//===>
//
//2 Bandy kierunek zgodny
VERSION : 0.1
VAR
  Banda_7 : FB 33;
  Banda_8 : FB 33;
END_VAR
VAR_TEMP
  Help_Bit_1 : BOOL ;
  Help_Reczny : BOOL ;
  Help_int : INT ;
  Help_Dword : DWORD ;
  Help_INT_1 : DINT ;
END_VAR
BEGIN
NETWORK
TITLE =
//Ten Network celowo jest wolny
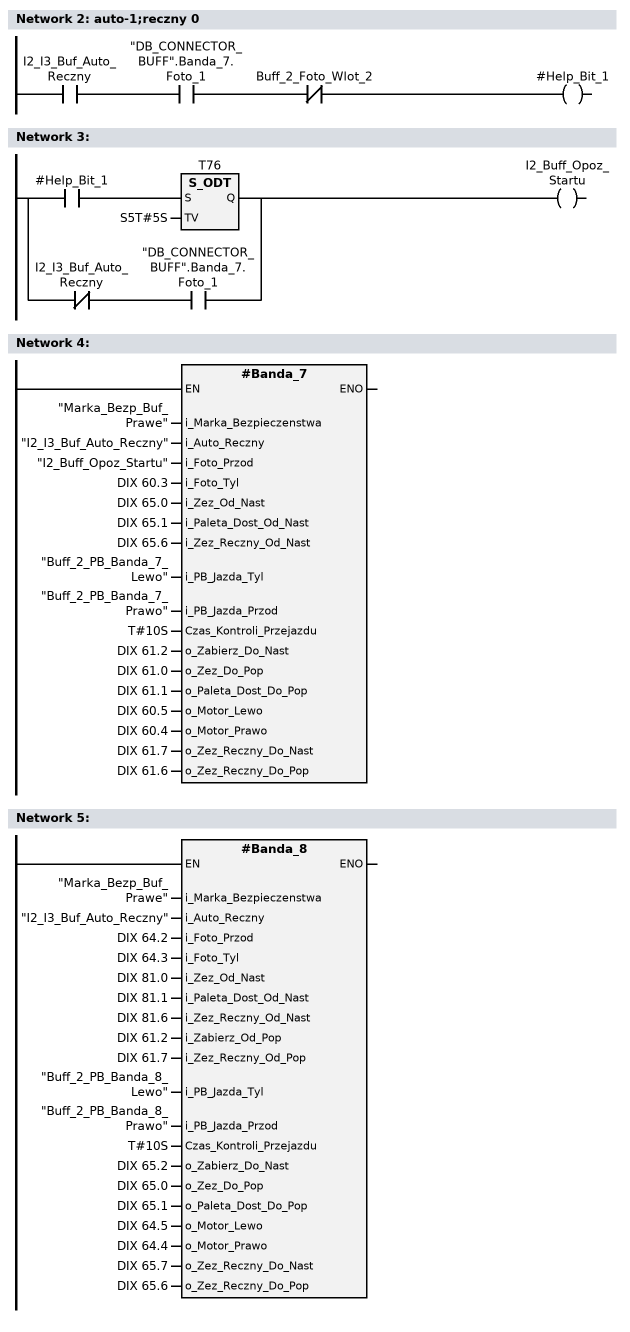
NETWORK
TITLE = auto-1;reczny 0
      A     "I2_I3_Buf_Auto_Reczny";
      A     "DB_CONNECTOR_BUFF".Banda_7.Foto_1;
      AN    "Buff_2_Foto_Wlot_2";
      =     #Help_Bit_1;
NETWORK
TITLE =
//Opoznienie startu po polozeniu palety
//
      O(;
      A     #Help_Bit_1;
      L     S5T#5S;
      SD    "T76";
      NOP   0;
      NOP   0;
      NOP   0;
      A     "T76";
      );
      O;
      AN    "I2_I3_Buf_Auto_Reczny";
      A     "DB_CONNECTOR_BUFF".Banda_7.Foto_1;
      =     "I2_Buff_Opoz_Startu";
NETWORK
TITLE =
//Banda 7
      CALL  #Banda_7 (
           i_Marka_Bezpieczenstwa   := "Marka_Bezp_Buf_Prawe",
           i_Auto_Reczny            := "I2_I3_Buf_Auto_Reczny",
           i_Foto_Przod             := "I2_Buff_Opoz_Startu",
           i_Foto_Tyl               := DIX 60.3,
           i_Zez_Od_Nast            := DIX 65.0,
           i_Paleta_Dost_Od_Nast    := DIX 65.1,
           i_Zez_Reczny_Od_Nast     := DIX 65.6,
           i_PB_Jazda_Tyl           := "Buff_2_PB_Banda_7_Lewo",
           i_PB_Jazda_Przod         := "Buff_2_PB_Banda_7_Prawo",
           Czas_Kontroli_Przejazdu  := T#10S,
           o_Zabierz_Do_Nast        := DIX 61.2,
           o_Zez_Do_Pop             := DIX 61.0,
           o_Paleta_Dost_Do_Pop     := DIX 61.1,
           o_Motor_Lewo             := DIX 60.5,
           o_Motor_Prawo            := DIX 60.4,
           o_Zez_Reczny_Do_Nast     := DIX 61.7,
           o_Zez_Reczny_Do_Pop      := DIX 61.6);
NETWORK
TITLE =
//Banda 8
      CALL  #Banda_8 (
           i_Marka_Bezpieczenstwa   := "Marka_Bezp_Buf_Prawe",
           i_Auto_Reczny            := "I2_I3_Buf_Auto_Reczny",
           i_Foto_Przod             := DIX 64.2,
           i_Foto_Tyl               := DIX 64.3,
           i_Zez_Od_Nast            := DIX 81.0,
           i_Paleta_Dost_Od_Nast    := DIX 81.1,
           i_Zez_Reczny_Od_Nast     := DIX 81.6,
           i_Zabierz_Od_Pop         := DIX 61.2,
           i_Zez_Reczny_Od_Pop      := DIX 61.7,
           i_PB_Jazda_Tyl           := "Buff_2_PB_Banda_8_Lewo",
           i_PB_Jazda_Przod         := "Buff_2_PB_Banda_8_Prawo",
           Czas_Kontroli_Przejazdu  := T#10S,
           o_Zabierz_Do_Nast        := DIX 65.2,
           o_Zez_Do_Pop             := DIX 65.0,
           o_Paleta_Dost_Do_Pop     := DIX 65.1,
           o_Motor_Lewo             := DIX 64.5,
           o_Motor_Prawo            := DIX 64.4,
           o_Zez_Reczny_Do_Nast     := DIX 65.7,
           o_Zez_Reczny_Do_Pop      := DIX 65.6);
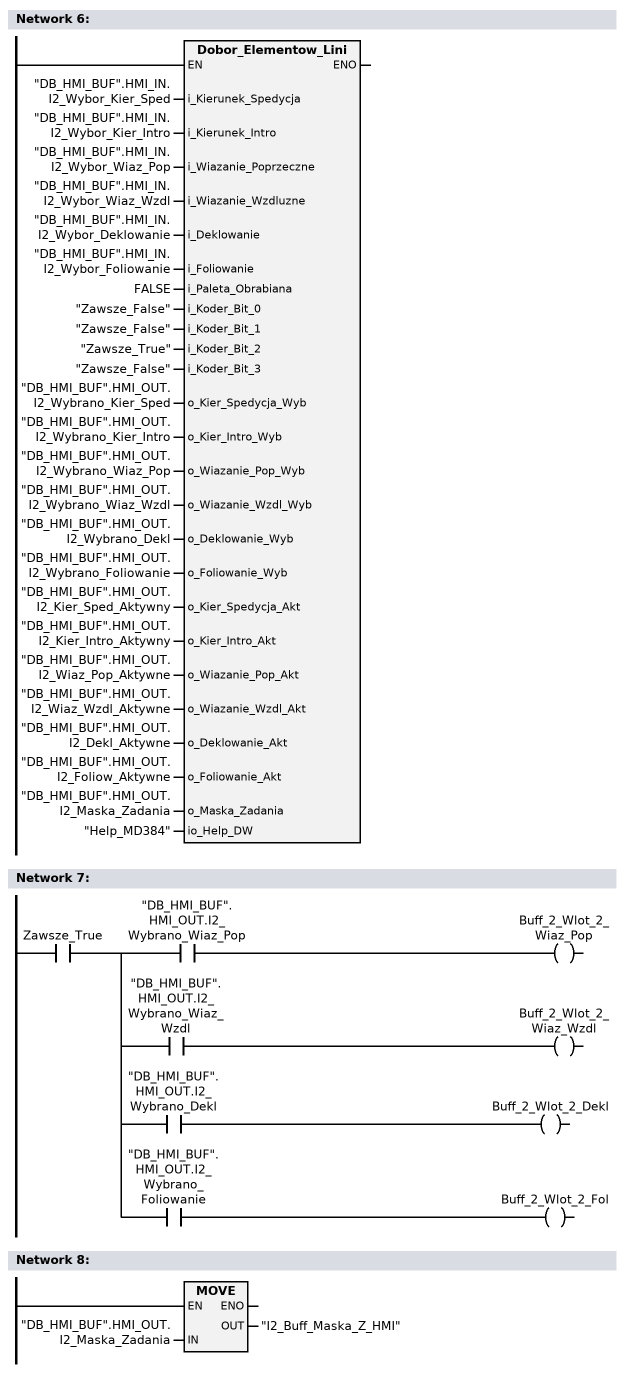
NETWORK
TITLE =
//Wybor Elementow na lini koder nr 4
      CALL  "Dobor_Elementow_Lini" (
           i_Kierunek_Spedycja      := "DB_HMI_BUF".HMI_IN.I2_Wybor_Kier_Sped,
           i_Kierunek_Intro         := "DB_HMI_BUF".HMI_IN.I2_Wybor_Kier_Intro,
           i_Wiazanie_Poprzeczne    := "DB_HMI_BUF".HMI_IN.I2_Wybor_Wiaz_Pop,
           i_Wiazanie_Wzdluzne      := "DB_HMI_BUF".HMI_IN.I2_Wybor_Wiaz_Wzdl,
           i_Deklowanie             := "DB_HMI_BUF".HMI_IN.I2_Wybor_Deklowanie,
           i_Foliowanie             := "DB_HMI_BUF".HMI_IN.I2_Wybor_Foliowanie,
           i_Paleta_Obrabiana       := FALSE,
           i_Koder_Bit_0            := "Zawsze_False",
           i_Koder_Bit_1            := "Zawsze_False",
           i_Koder_Bit_2            := "Zawsze_True",
           i_Koder_Bit_3            := "Zawsze_False",
           o_Kier_Spedycja_Wyb      := "DB_HMI_BUF".HMI_OUT.I2_Wybrano_Kier_Sped,
           o_Kier_Intro_Wyb         := "DB_HMI_BUF".HMI_OUT.I2_Wybrano_Kier_Intro,
           o_Wiazanie_Pop_Wyb       := "DB_HMI_BUF".HMI_OUT.I2_Wybrano_Wiaz_Pop,
           o_Wiazanie_Wzdl_Wyb      := "DB_HMI_BUF".HMI_OUT.I2_Wybrano_Wiaz_Wzdl,
           o_Deklowanie_Wyb         := "DB_HMI_BUF".HMI_OUT.I2_Wybrano_Dekl,
           o_Foliowanie_Wyb         := "DB_HMI_BUF".HMI_OUT.I2_Wybrano_Foliowanie,
           o_Kier_Spedycja_Akt      := "DB_HMI_BUF".HMI_OUT.I2_Kier_Sped_Aktywny,
           o_Kier_Intro_Akt         := "DB_HMI_BUF".HMI_OUT.I2_Kier_Intro_Aktywny,
           o_Wiazanie_Pop_Akt       := "DB_HMI_BUF".HMI_OUT.I2_Wiaz_Pop_Aktywne,
           o_Wiazanie_Wzdl_Akt      := "DB_HMI_BUF".HMI_OUT.I2_Wiaz_Wzdl_Aktywne,
           o_Deklowanie_Akt         := "DB_HMI_BUF".HMI_OUT.I2_Dekl_Aktywne,
           o_Foliowanie_Akt         := "DB_HMI_BUF".HMI_OUT.I2_Foliow_Aktywne,
           o_Maska_Zadania          := "DB_HMI_BUF".HMI_OUT.I2_Maska_Zadania,
           io_Help_DW               := "Help_MD384");
NETWORK
TITLE =
//Wyswietlenie lampek zadania lini
      A     "Zawsze_True";
      =     L 12.0;
      A     L 12.0;
      A     "DB_HMI_BUF".HMI_OUT.I2_Wybrano_Wiaz_Pop;
      =     "Buff_2_Wlot_2_Wiaz_Pop";
      A     L 12.0;
      A     "DB_HMI_BUF".HMI_OUT.I2_Wybrano_Wiaz_Wzdl;
      =     "Buff_2_Wlot_2_Wiaz_Wzdl";
      A     L 12.0;
      A     "DB_HMI_BUF".HMI_OUT.I2_Wybrano_Dekl;
      =     "Buff_2_Wlot_2_Dekl";
      A     L 12.0;
      A     "DB_HMI_BUF".HMI_OUT.I2_Wybrano_Foliowanie;
      =     "Buff_2_Wlot_2_Fol";
NETWORK
TITLE =
//Przypisanie maski zadania do bandy wejsciowej
      L     "DB_HMI_BUF".HMI_OUT.I2_Maska_Zadania;
      T     "I2_Buff_Maska_Z_HMI";
      NOP   0;
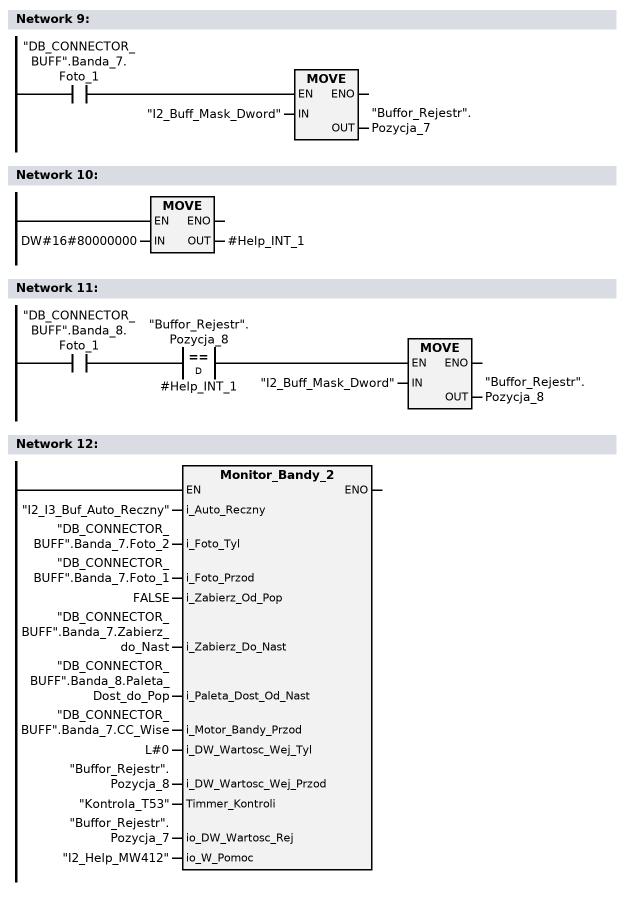
NETWORK
TITLE =
//Zbudowanie z maski podwojnego slowa
      A     "DB_CONNECTOR_BUFF".Banda_7.Foto_1;
      JNB   _001;
      L     "I2_Buff_Mask_Dword";
      T     "Buffor_Rejestr".Pozycja_7;
_001: NOP   0;
NETWORK
TITLE =
      L     DW#16#80000000;
      T     #Help_INT_1;
      NOP   0;
NETWORK
TITLE =
//sprawdzenie dla fotokomorki bandy 8
      A     "DB_CONNECTOR_BUFF".Banda_8.Foto_1;
      A(;
      L     "Buffor_Rejestr".Pozycja_8;
      L     #Help_INT_1;
      ==D;
      );
      JNB   _002;
      L     "I2_Buff_Mask_Dword";
      T     "Buffor_Rejestr".Pozycja_8;
_002: NOP   0;
NETWORK
TITLE =
//Monitoring band 7
      CALL  "Monitor_Bandy_2" (
           i_Auto_Reczny            := "I2_I3_Buf_Auto_Reczny",
           i_Foto_Tyl               := "DB_CONNECTOR_BUFF".Banda_7.Foto_2,
           i_Foto_Przod             := "DB_CONNECTOR_BUFF".Banda_7.Foto_1,
           i_Zabierz_Od_Pop         := FALSE,
           i_Zabierz_Do_Nast        := "DB_CONNECTOR_BUFF".Banda_7.Zabierz_do_Nast,
           i_Paleta_Dost_Od_Nast    := "DB_CONNECTOR_BUFF".Banda_8.Paleta_Dost_do_Pop,
           i_Motor_Bandy_Przod      := "DB_CONNECTOR_BUFF".Banda_7.CC_Wise,
           i_DW_Wartosc_Wej_Tyl     := L#0,
           i_DW_Wartosc_Wej_Przod   := "Buffor_Rejestr".Pozycja_8,
           Timmer_Kontroli          := "Kontrola_T53",
           io_DW_Wartosc_Rej        := "Buffor_Rejestr".Pozycja_7,
           io_W_Pomoc               := "I2_Help_MW412");
